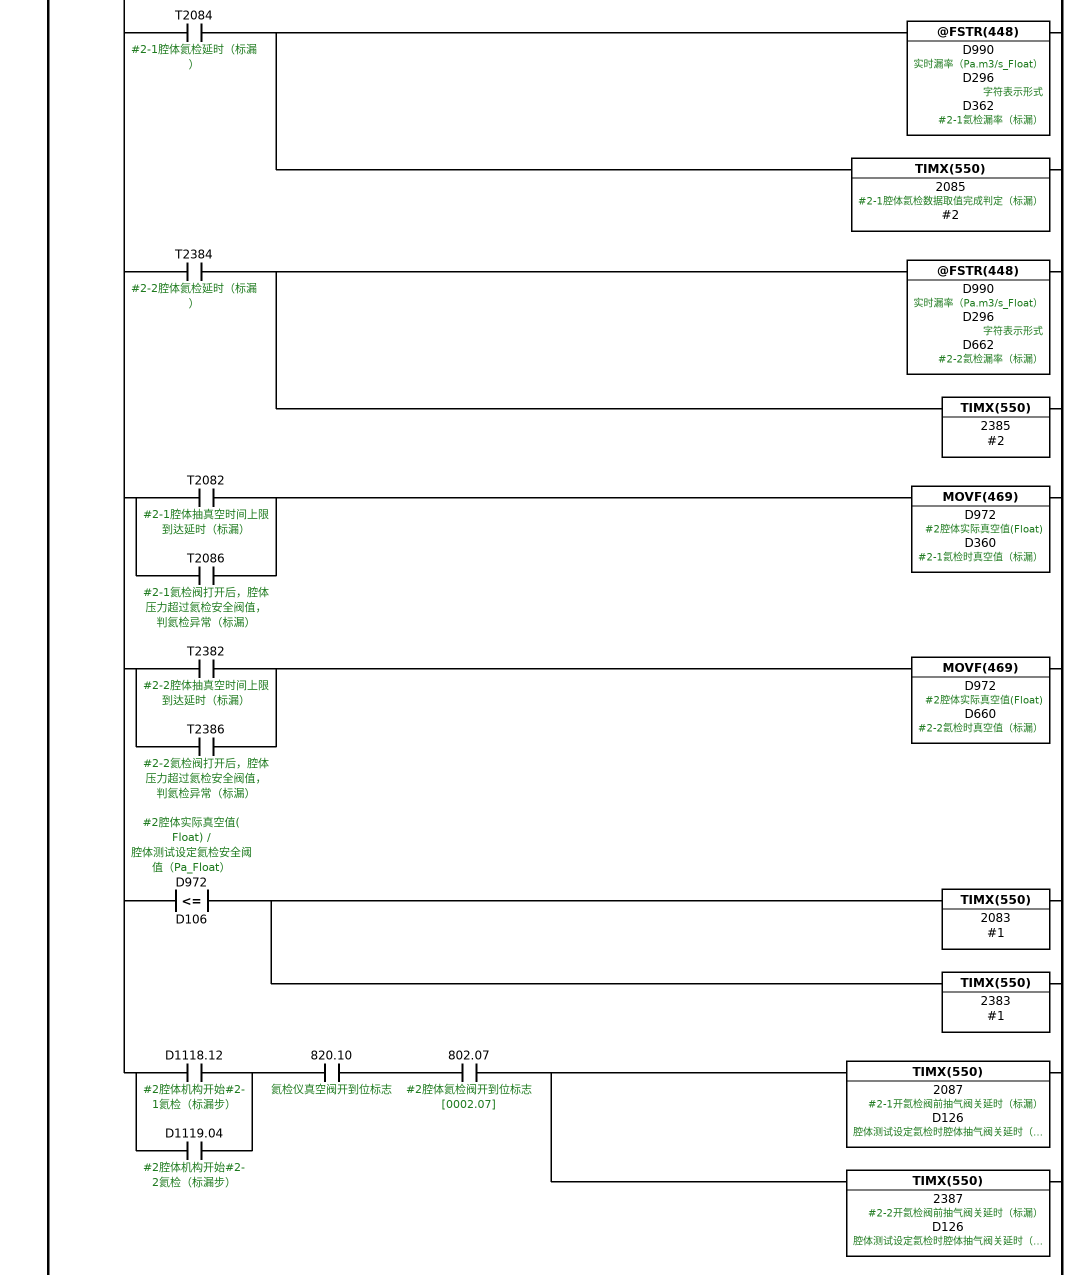
; rung 20: 标漏测试数据处理
LD P_On
OUT TR0
LD D1118.08  ; #2腔体机构开#2腔抽气阀（标漏步）
AND 821.10  ; #2-1腔体阀开到位标志
LD D1119.00  ; #2腔体机构开#2腔抽真空阀（标漏步）
AND 821.12  ; #2-2腔体阀开到位标志
ORLD
ANDLD
AND 821.08  ; #2腔体抽真空阀开到位标志
AND<=F(332) D972 D100  ; #2腔体实际真空值(Float), 腔体测试设定真空阈值（Pa_Float）
TIMX(550) 2081 #0  ; #2-1腔体抽真空阀值到达延时（标漏）
TIMX(550) 2381 #0  ; #2-2腔体抽真空阀值到达延时（标漏）
LD TR0
LD D1118.08  ; #2腔体机构开#2腔抽气阀（标漏步）
AND 821.10  ; #2-1腔体阀开到位标志
LD D1119.00  ; #2腔体机构开#2腔抽真空阀（标漏步）
AND 821.12  ; #2-2腔体阀开到位标志
ORLD
ANDLD
AND 821.08  ; #2腔体抽真空阀开到位标志
AND>F(333) D972 D100  ; #2腔体实际真空值(Float), 腔体测试设定真空阈值（Pa_Float）
TIMX(550) 2082 D102  ; 腔体测试设定抽真空时间上限（S_UInt）, #2-1腔体抽真空时间上限到达延时（标漏）
TIMX(550) 2382 D102  ; 腔体测试设定抽真空时间上限（S_UInt）, #2-2腔体抽真空时间上限到达延时（标漏）
LD TR0
AND D1118.12  ; #2腔体机构开始#2-1氦检（标漏步）
AND 821.10  ; #2-1腔体阀开到位标志
AND 820.10  ; 氦检仪真空阀开到位标志
AND 802.07  ; #2腔体氦检阀开到位标志[0002.07]
TIMX(550) 2084 D110  ; 腔体测试设定氦检时间（S_UInt）, #2-1腔体氦检延时（标漏）
@MOVF(469) D972 D360  ; #2腔体实际真空值(Float), #2-1氦检时真空值（标漏）
AND>F(333) D972 D106  ; #2腔体实际真空值(Float), 腔体测试设定氦检安全阈值（Pa_Float）
TIMX(550) 2086 #0  ; #2-1氦检阀打开后，腔体压力超过氦检安全阀值，判氦检异常（标漏）
LD TR0
AND D1119.04  ; #2腔体机构开始#2-2氦检（标漏步）
AND 821.12  ; #2-2腔体阀开到位标志
AND 820.10  ; 氦检仪真空阀开到位标志
AND 802.07  ; #2腔体氦检阀开到位标志[0002.07]
TIMX(550) 2384 D110  ; 腔体测试设定氦检时间（S_UInt）, #2-2腔体氦检延时（标漏）
@MOVF(469) D972 D660  ; #2腔体实际真空值(Float), #2-2氦检时真空值（标漏）
AND>F(333) D972 D106  ; #2腔体实际真空值(Float), 腔体测试设定氦检安全阈值（Pa_Float）
TIMX(550) 2386 #0  ; #2-2氦检阀打开后，腔体压力超过氦检安全阀值，判氦检异常（标漏）
LD TR0
AND T2084  ; #2-1腔体氦检延时（标漏）
@FSTR(448) D990 D296 D362  ; 实时漏率（Pa.m3/s_Float）, 字符表示形式, #2-1氦检漏率（标漏）
TIMX(550) 2085 #2  ; #2-1腔体氦检数据取值完成判定（标漏）
LD TR0
AND T2384  ; #2-2腔体氦检延时（标漏）
@FSTR(448) D990 D296 D662  ; 实时漏率（Pa.m3/s_Float）, 字符表示形式, #2-2氦检漏率（标漏）
TIMX(550) 2385 #2
LD TR0
LD T2082  ; #2-1腔体抽真空时间上限到达延时（标漏）
OR T2086  ; #2-1氦检阀打开后，腔体压力超过氦检安全阀值，判氦检异常（标漏）
ANDLD
MOVF(469) D972 D360  ; #2腔体实际真空值(Float), #2-1氦检时真空值（标漏）
LD TR0
LD T2382  ; #2-2腔体抽真空时间上限到达延时（标漏）
OR T2386  ; #2-2氦检阀打开后，腔体压力超过氦检安全阀值，判氦检异常（标漏）
ANDLD
MOVF(469) D972 D660  ; #2腔体实际真空值(Float), #2-2氦检时真空值（标漏）
LD TR0
AND<=F(332) D972 D106  ; #2腔体实际真空值(Float), 腔体测试设定氦检安全阈值（Pa_Float）
TIMX(550) 2083 #1
TIMX(550) 2383 #1
LD TR0
LD D1118.12  ; #2腔体机构开始#2-1氦检（标漏步）
OR D1119.04  ; #2腔体机构开始#2-2氦检（标漏步）
ANDLD
AND 820.10  ; 氦检仪真空阀开到位标志
AND 802.07  ; #2腔体氦检阀开到位标志[0002.07]
TIMX(550) 2087 D126  ; 腔体测试设定氦检时腔体抽气阀关延时（S_UInt）, #2-1开氦检阀前抽气阀关延时（标漏）
TIMX(550) 2387 D126  ; 腔体测试设定氦检时腔体抽气阀关延时（S_UInt）, #2-2开氦检阀前抽气阀关延时（标漏）
; rung 21: ********************** / #3腔体标漏流程 / **********************

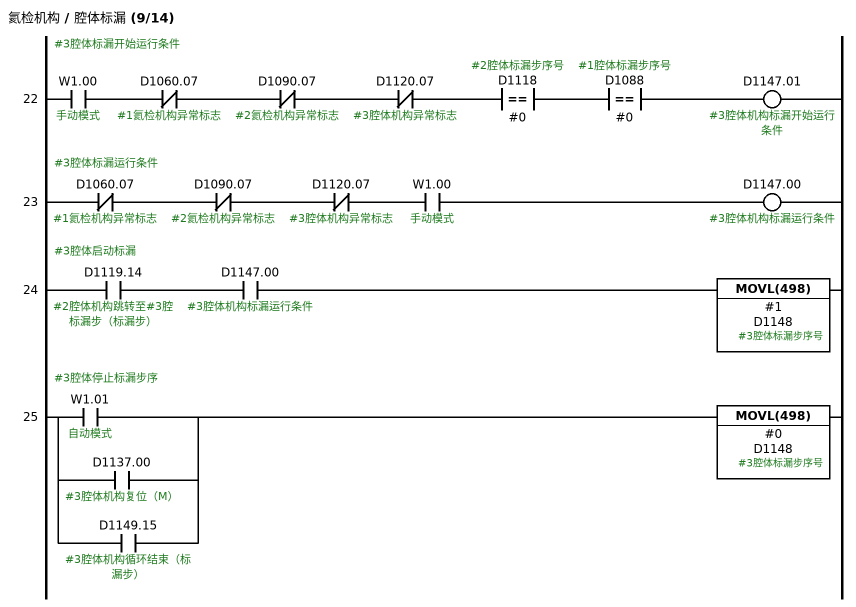
; rung 22: #3腔体标漏开始运行条件
LD W1.00  ; 手动模式
ANDNOT D1060.07  ; #1氦检机构异常标志
ANDNOT D1090.07  ; #2氦检机构异常标志
ANDNOT D1120.07  ; #3腔体机构异常标志
AND=L(301) D1118 #0  ; #2腔体标漏步序号
AND=L(301) D1088 #0  ; #1腔体标漏步序号
OUT D1147.01  ; #3腔体机构标漏开始运行条件
; rung 23: #3腔体标漏运行条件
LDNOT D1060.07  ; #1氦检机构异常标志
ANDNOT D1090.07  ; #2氦检机构异常标志
ANDNOT D1120.07  ; #3腔体机构异常标志
AND W1.00  ; 手动模式
OUT D1147.00  ; #3腔体机构标漏运行条件
; rung 24: #3腔体启动标漏
LD D1119.14  ; #2腔体机构跳转至#3腔标漏步（标漏步）
AND D1147.00  ; #3腔体机构标漏运行条件
MOVL(498) #1 D1148  ; #3腔体标漏步序号
; rung 25: #3腔体停止标漏步序
LD W1.01  ; 自动模式
OR D1137.00  ; #3腔体机构复位（M）
OR D1149.15  ; #3腔体机构循环结束（标漏步）
MOVL(498) #0 D1148  ; #3腔体标漏步序号

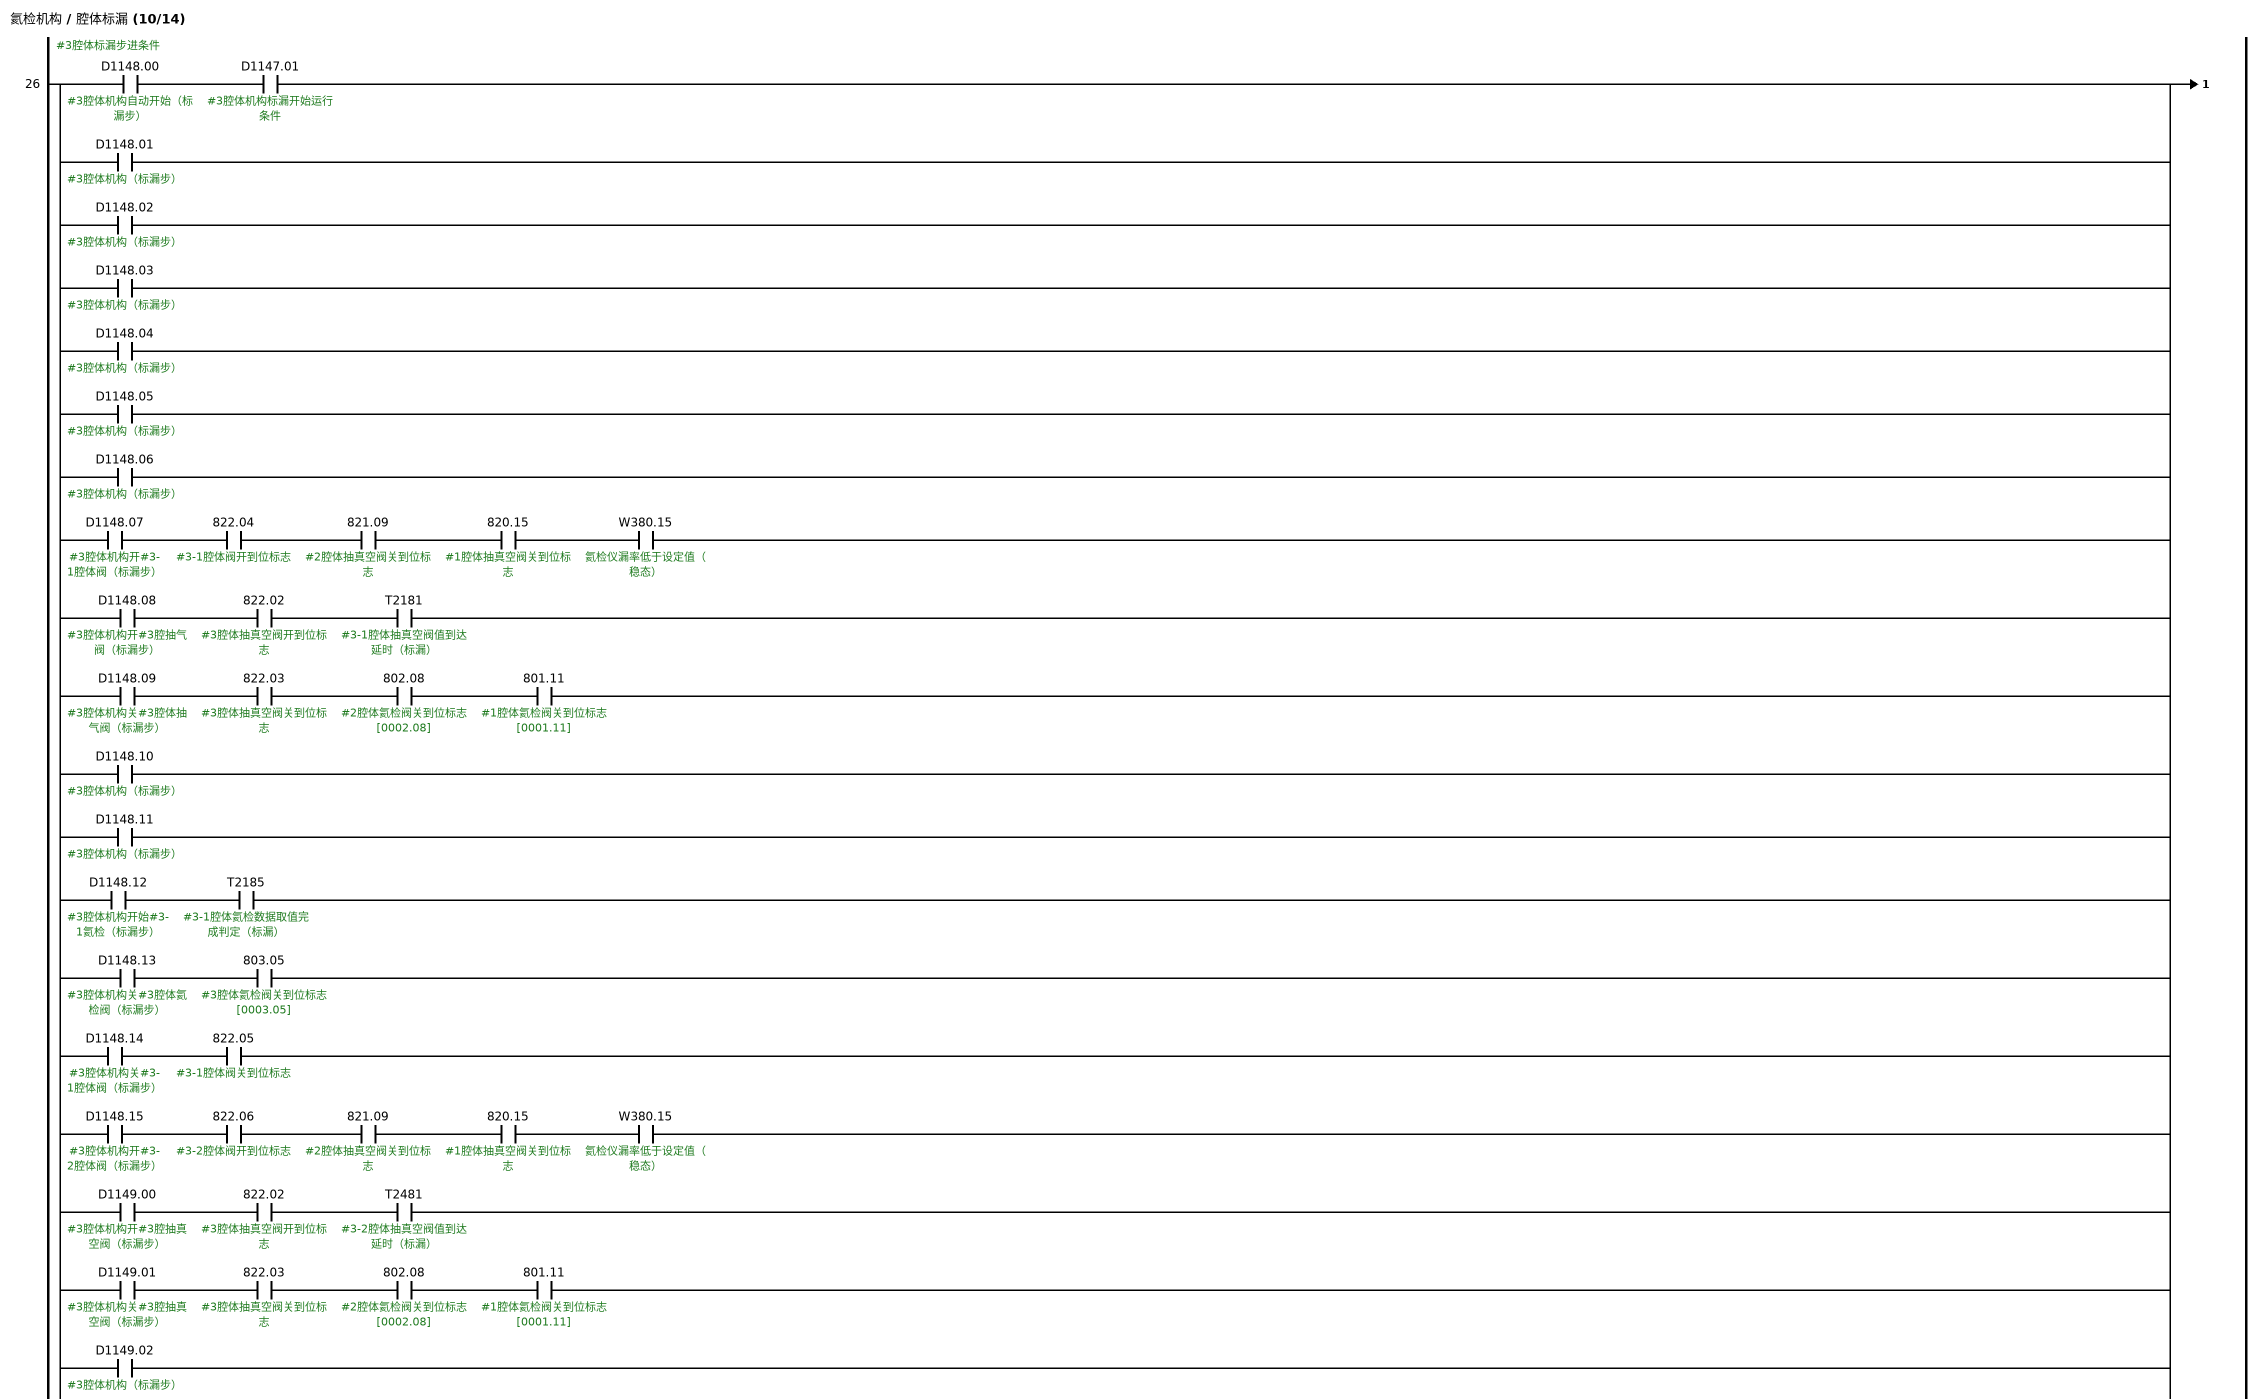

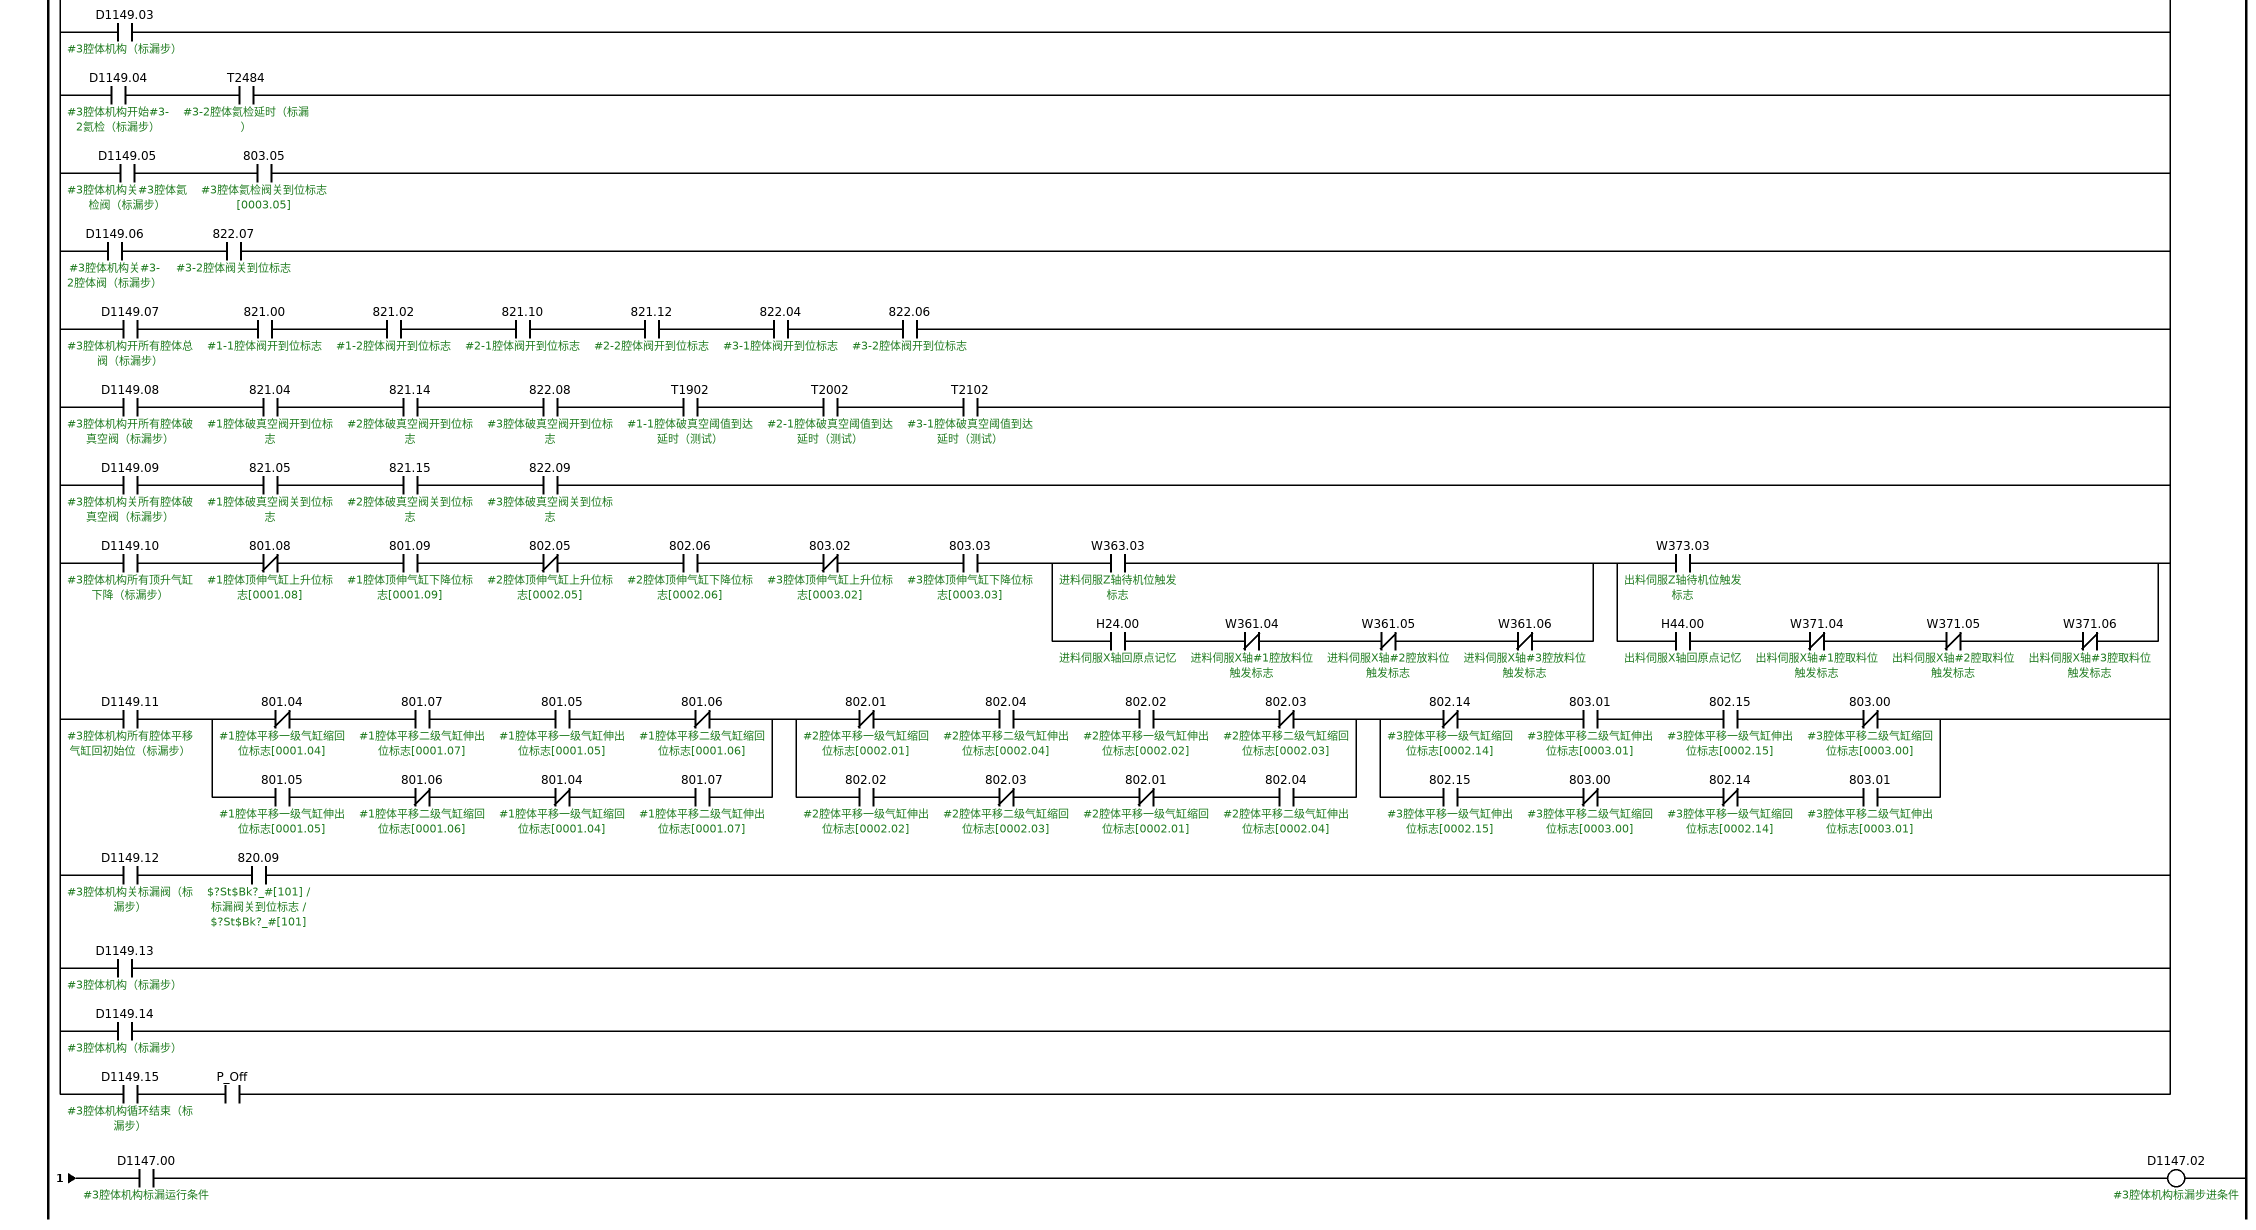
; rung 26: #3腔体标漏步进条件
LD D1148.00  ; #3腔体机构自动开始（标漏步）
AND D1147.01  ; #3腔体机构标漏开始运行条件
OR D1148.01  ; #3腔体机构（标漏步）
OR D1148.02  ; #3腔体机构（标漏步）
OR D1148.03  ; #3腔体机构（标漏步）
OR D1148.04  ; #3腔体机构（标漏步）
OR D1148.05  ; #3腔体机构（标漏步）
OR D1148.06  ; #3腔体机构（标漏步）
LD D1148.07  ; #3腔体机构开#3-1腔体阀（标漏步）
AND 822.04  ; #3-1腔体阀开到位标志
AND 821.09  ; #2腔体抽真空阀关到位标志
AND 820.15  ; #1腔体抽真空阀关到位标志
AND W380.15  ; 氦检仪漏率低于设定值（稳态）
ORLD
LD D1148.08  ; #3腔体机构开#3腔抽气阀（标漏步）
AND 822.02  ; #3腔体抽真空阀开到位标志
AND T2181  ; #3-1腔体抽真空阀值到达延时（标漏）
ORLD
LD D1148.09  ; #3腔体机构关#3腔体抽气阀（标漏步）
AND 822.03  ; #3腔体抽真空阀关到位标志
AND 802.08  ; #2腔体氦检阀关到位标志[0002.08]
AND 801.11  ; #1腔体氦检阀关到位标志[0001.11]
ORLD
OR D1148.10  ; #3腔体机构（标漏步）
OR D1148.11  ; #3腔体机构（标漏步）
LD D1148.12  ; #3腔体机构开始#3-1氦检（标漏步）
AND T2185  ; #3-1腔体氦检数据取值完成判定（标漏）
ORLD
LD D1148.13  ; #3腔体机构关#3腔体氦检阀（标漏步）
AND 803.05  ; #3腔体氦检阀关到位标志[0003.05]
ORLD
LD D1148.14  ; #3腔体机构关#3-1腔体阀（标漏步）
AND 822.05  ; #3-1腔体阀关到位标志
ORLD
LD D1148.15  ; #3腔体机构开#3-2腔体阀（标漏步）
AND 822.06  ; #3-2腔体阀开到位标志
AND 821.09  ; #2腔体抽真空阀关到位标志
AND 820.15  ; #1腔体抽真空阀关到位标志
AND W380.15  ; 氦检仪漏率低于设定值（稳态）
ORLD
LD D1149.00  ; #3腔体机构开#3腔抽真空阀（标漏步）
AND 822.02  ; #3腔体抽真空阀开到位标志
AND T2481  ; #3-2腔体抽真空阀值到达延时（标漏）
ORLD
LD D1149.01  ; #3腔体机构关#3腔抽真空阀（标漏步）
AND 822.03  ; #3腔体抽真空阀关到位标志
AND 802.08  ; #2腔体氦检阀关到位标志[0002.08]
AND 801.11  ; #1腔体氦检阀关到位标志[0001.11]
ORLD
OR D1149.02  ; #3腔体机构（标漏步）
OR D1149.03  ; #3腔体机构（标漏步）
LD D1149.04  ; #3腔体机构开始#3-2氦检（标漏步）
AND T2484  ; #3-2腔体氦检延时（标漏）
ORLD
LD D1149.05  ; #3腔体机构关#3腔体氦检阀（标漏步）
AND 803.05  ; #3腔体氦检阀关到位标志[0003.05]
ORLD
LD D1149.06  ; #3腔体机构关#3-2腔体阀（标漏步）
AND 822.07  ; #3-2腔体阀关到位标志
ORLD
LD D1149.07  ; #3腔体机构开所有腔体总阀（标漏步）
AND 821.00  ; #1-1腔体阀开到位标志
AND 821.02  ; #1-2腔体阀开到位标志
AND 821.10  ; #2-1腔体阀开到位标志
AND 821.12  ; #2-2腔体阀开到位标志
AND 822.04  ; #3-1腔体阀开到位标志
AND 822.06  ; #3-2腔体阀开到位标志
ORLD
LD D1149.08  ; #3腔体机构开所有腔体破真空阀（标漏步）
AND 821.04  ; #1腔体破真空阀开到位标志
AND 821.14  ; #2腔体破真空阀开到位标志
AND 822.08  ; #3腔体破真空阀开到位标志
AND T1902  ; #1-1腔体破真空阈值到达延时（测试）
AND T2002  ; #2-1腔体破真空阈值到达延时（测试）
AND T2102  ; #3-1腔体破真空阈值到达延时（测试）
ORLD
LD D1149.09  ; #3腔体机构关所有腔体破真空阀（标漏步）
AND 821.05  ; #1腔体破真空阀关到位标志
AND 821.15  ; #2腔体破真空阀关到位标志
AND 822.09  ; #3腔体破真空阀关到位标志
ORLD
LD D1149.10  ; #3腔体机构所有顶升气缸下降（标漏步）
ANDNOT 801.08  ; #1腔体顶伸气缸上升位标志[0001.08]
AND 801.09  ; #1腔体顶伸气缸下降位标志[0001.09]
ANDNOT 802.05  ; #2腔体顶伸气缸上升位标志[0002.05]
AND 802.06  ; #2腔体顶伸气缸下降位标志[0002.06]
ANDNOT 803.02  ; #3腔体顶伸气缸上升位标志[0003.02]
AND 803.03  ; #3腔体顶伸气缸下降位标志[0003.03]
LD W363.03  ; 进料伺服Z轴待机位触发标志
LD H24.00  ; 进料伺服X轴回原点记忆
ANDNOT W361.04  ; 进料伺服X轴#1腔放料位触发标志
ANDNOT W361.05  ; 进料伺服X轴#2腔放料位触发标志
ANDNOT W361.06  ; 进料伺服X轴#3腔放料位触发标志
ORLD
ANDLD
LD W373.03  ; 出料伺服Z轴待机位触发标志
LD H44.00  ; 出料伺服X轴回原点记忆
ANDNOT W371.04  ; 出料伺服X轴#1腔取料位触发标志
ANDNOT W371.05  ; 出料伺服X轴#2腔取料位触发标志
ANDNOT W371.06  ; 出料伺服X轴#3腔取料位触发标志
ORLD
ANDLD
ORLD
LD D1149.11  ; #3腔体机构所有腔体平移气缸回初始位（标漏步）
LDNOT 801.04  ; #1腔体平移一级气缸缩回位标志[0001.04]
AND 801.07  ; #1腔体平移二级气缸伸出位标志[0001.07]
AND 801.05  ; #1腔体平移一级气缸伸出位标志[0001.05]
ANDNOT 801.06  ; #1腔体平移二级气缸缩回位标志[0001.06]
LD 801.05  ; #1腔体平移一级气缸伸出位标志[0001.05]
ANDNOT 801.06  ; #1腔体平移二级气缸缩回位标志[0001.06]
ANDNOT 801.04  ; #1腔体平移一级气缸缩回位标志[0001.04]
AND 801.07  ; #1腔体平移二级气缸伸出位标志[0001.07]
ORLD
ANDLD
LDNOT 802.01  ; #2腔体平移一级气缸缩回位标志[0002.01]
AND 802.04  ; #2腔体平移二级气缸伸出位标志[0002.04]
AND 802.02  ; #2腔体平移一级气缸伸出位标志[0002.02]
ANDNOT 802.03  ; #2腔体平移二级气缸缩回位标志[0002.03]
LD 802.02  ; #2腔体平移一级气缸伸出位标志[0002.02]
ANDNOT 802.03  ; #2腔体平移二级气缸缩回位标志[0002.03]
ANDNOT 802.01  ; #2腔体平移一级气缸缩回位标志[0002.01]
AND 802.04  ; #2腔体平移二级气缸伸出位标志[0002.04]
ORLD
ANDLD
LDNOT 802.14  ; #3腔体平移一级气缸缩回位标志[0002.14]
AND 803.01  ; #3腔体平移二级气缸伸出位标志[0003.01]
AND 802.15  ; #3腔体平移一级气缸伸出位标志[0002.15]
ANDNOT 803.00  ; #3腔体平移二级气缸缩回位标志[0003.00]
LD 802.15  ; #3腔体平移一级气缸伸出位标志[0002.15]
ANDNOT 803.00  ; #3腔体平移二级气缸缩回位标志[0003.00]
ANDNOT 802.14  ; #3腔体平移一级气缸缩回位标志[0002.14]
AND 803.01  ; #3腔体平移二级气缸伸出位标志[0003.01]
ORLD
ANDLD
ORLD
LD D1149.12  ; #3腔体机构关标漏阀（标漏步）
AND 820.09  ; $?St$Bk?_#[101] / 标漏阀关到位标志 / $?St$Bk?_#[101]
ORLD
OR D1149.13  ; #3腔体机构（标漏步）
OR D1149.14  ; #3腔体机构（标漏步）
LD D1149.15  ; #3腔体机构循环结束（标漏步）
AND P_Off
ORLD
AND D1147.00  ; #3腔体机构标漏运行条件
OUT D1147.02  ; #3腔体机构标漏步进条件

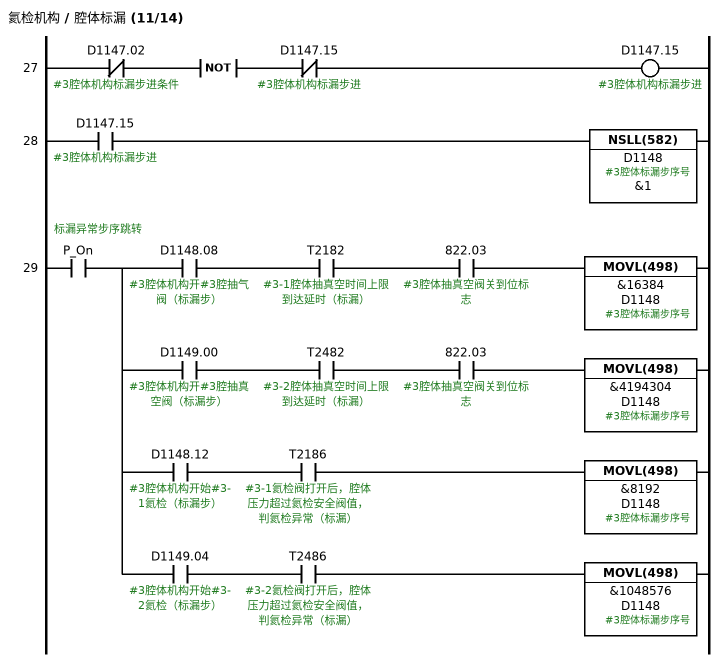
; rung 27
LDNOT D1147.02  ; #3腔体机构标漏步进条件
NOT(520)
ANDNOT D1147.15  ; #3腔体机构标漏步进
OUT D1147.15  ; #3腔体机构标漏步进
; rung 28
LD D1147.15  ; #3腔体机构标漏步进
NSLL(582) D1148 &1  ; #3腔体标漏步序号
; rung 29: 标漏异常步序跳转
LD P_On
OUT TR0
AND D1148.08  ; #3腔体机构开#3腔抽气阀（标漏步）
AND T2182  ; #3-1腔体抽真空时间上限到达延时（标漏）
AND 822.03  ; #3腔体抽真空阀关到位标志
MOVL(498) &16384 D1148  ; #3腔体标漏步序号
LD TR0
AND D1149.00  ; #3腔体机构开#3腔抽真空阀（标漏步）
AND T2482  ; #3-2腔体抽真空时间上限到达延时（标漏）
AND 822.03  ; #3腔体抽真空阀关到位标志
MOVL(498) &4194304 D1148  ; #3腔体标漏步序号
LD TR0
AND D1148.12  ; #3腔体机构开始#3-1氦检（标漏步）
AND T2186  ; #3-1氦检阀打开后，腔体压力超过氦检安全阀值，判氦检异常（标漏）
MOVL(498) &8192 D1148  ; #3腔体标漏步序号
LD TR0
AND D1149.04  ; #3腔体机构开始#3-2氦检（标漏步）
AND T2486  ; #3-2氦检阀打开后，腔体压力超过氦检安全阀值，判氦检异常（标漏）
MOVL(498) &1048576 D1148  ; #3腔体标漏步序号

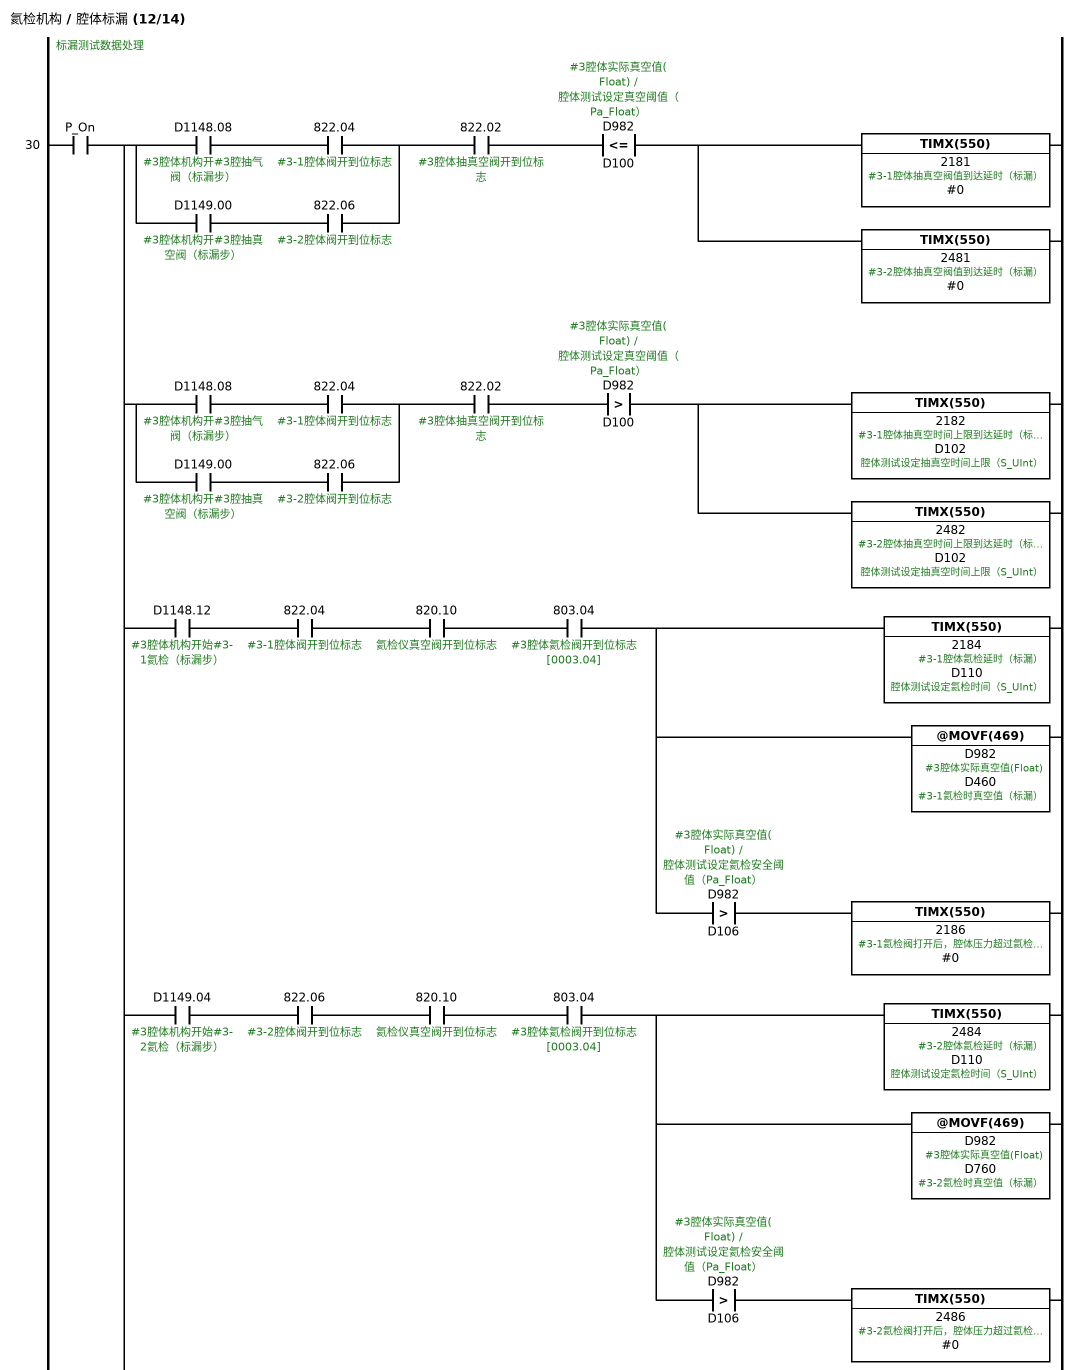

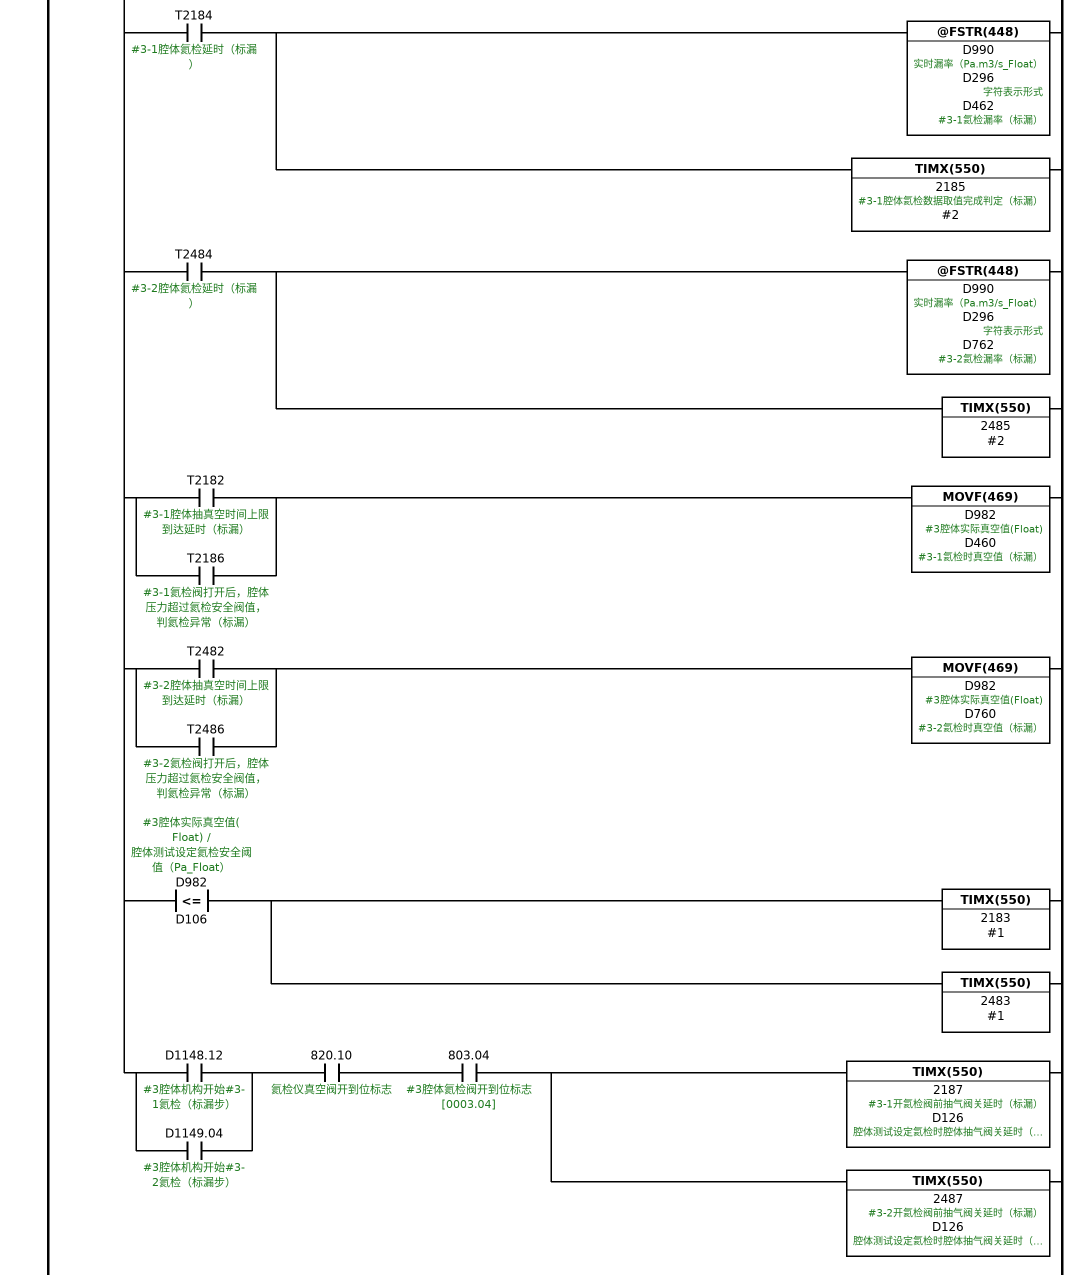
; rung 30: 标漏测试数据处理
LD P_On
OUT TR0
LD D1148.08  ; #3腔体机构开#3腔抽气阀（标漏步）
AND 822.04  ; #3-1腔体阀开到位标志
LD D1149.00  ; #3腔体机构开#3腔抽真空阀（标漏步）
AND 822.06  ; #3-2腔体阀开到位标志
ORLD
ANDLD
AND 822.02  ; #3腔体抽真空阀开到位标志
AND<=F(332) D982 D100  ; #3腔体实际真空值(Float), 腔体测试设定真空阈值（Pa_Float）
TIMX(550) 2181 #0  ; #3-1腔体抽真空阀值到达延时（标漏）
TIMX(550) 2481 #0  ; #3-2腔体抽真空阀值到达延时（标漏）
LD TR0
LD D1148.08  ; #3腔体机构开#3腔抽气阀（标漏步）
AND 822.04  ; #3-1腔体阀开到位标志
LD D1149.00  ; #3腔体机构开#3腔抽真空阀（标漏步）
AND 822.06  ; #3-2腔体阀开到位标志
ORLD
ANDLD
AND 822.02  ; #3腔体抽真空阀开到位标志
AND>F(333) D982 D100  ; #3腔体实际真空值(Float), 腔体测试设定真空阈值（Pa_Float）
TIMX(550) 2182 D102  ; 腔体测试设定抽真空时间上限（S_UInt）, #3-1腔体抽真空时间上限到达延时（标漏）
TIMX(550) 2482 D102  ; 腔体测试设定抽真空时间上限（S_UInt）, #3-2腔体抽真空时间上限到达延时（标漏）
LD TR0
AND D1148.12  ; #3腔体机构开始#3-1氦检（标漏步）
AND 822.04  ; #3-1腔体阀开到位标志
AND 820.10  ; 氦检仪真空阀开到位标志
AND 803.04  ; #3腔体氦检阀开到位标志[0003.04]
TIMX(550) 2184 D110  ; 腔体测试设定氦检时间（S_UInt）, #3-1腔体氦检延时（标漏）
@MOVF(469) D982 D460  ; #3腔体实际真空值(Float), #3-1氦检时真空值（标漏）
AND>F(333) D982 D106  ; #3腔体实际真空值(Float), 腔体测试设定氦检安全阈值（Pa_Float）
TIMX(550) 2186 #0  ; #3-1氦检阀打开后，腔体压力超过氦检安全阀值，判氦检异常（标漏）
LD TR0
AND D1149.04  ; #3腔体机构开始#3-2氦检（标漏步）
AND 822.06  ; #3-2腔体阀开到位标志
AND 820.10  ; 氦检仪真空阀开到位标志
AND 803.04  ; #3腔体氦检阀开到位标志[0003.04]
TIMX(550) 2484 D110  ; 腔体测试设定氦检时间（S_UInt）, #3-2腔体氦检延时（标漏）
@MOVF(469) D982 D760  ; #3腔体实际真空值(Float), #3-2氦检时真空值（标漏）
AND>F(333) D982 D106  ; #3腔体实际真空值(Float), 腔体测试设定氦检安全阈值（Pa_Float）
TIMX(550) 2486 #0  ; #3-2氦检阀打开后，腔体压力超过氦检安全阀值，判氦检异常（标漏）
LD TR0
AND T2184  ; #3-1腔体氦检延时（标漏）
@FSTR(448) D990 D296 D462  ; 实时漏率（Pa.m3/s_Float）, 字符表示形式, #3-1氦检漏率（标漏）
TIMX(550) 2185 #2  ; #3-1腔体氦检数据取值完成判定（标漏）
LD TR0
AND T2484  ; #3-2腔体氦检延时（标漏）
@FSTR(448) D990 D296 D762  ; 实时漏率（Pa.m3/s_Float）, 字符表示形式, #3-2氦检漏率（标漏）
TIMX(550) 2485 #2
LD TR0
LD T2182  ; #3-1腔体抽真空时间上限到达延时（标漏）
OR T2186  ; #3-1氦检阀打开后，腔体压力超过氦检安全阀值，判氦检异常（标漏）
ANDLD
MOVF(469) D982 D460  ; #3腔体实际真空值(Float), #3-1氦检时真空值（标漏）
LD TR0
LD T2482  ; #3-2腔体抽真空时间上限到达延时（标漏）
OR T2486  ; #3-2氦检阀打开后，腔体压力超过氦检安全阀值，判氦检异常（标漏）
ANDLD
MOVF(469) D982 D760  ; #3腔体实际真空值(Float), #3-2氦检时真空值（标漏）
LD TR0
AND<=F(332) D982 D106  ; #3腔体实际真空值(Float), 腔体测试设定氦检安全阈值（Pa_Float）
TIMX(550) 2183 #1
TIMX(550) 2483 #1
LD TR0
LD D1148.12  ; #3腔体机构开始#3-1氦检（标漏步）
OR D1149.04  ; #3腔体机构开始#3-2氦检（标漏步）
ANDLD
AND 820.10  ; 氦检仪真空阀开到位标志
AND 803.04  ; #3腔体氦检阀开到位标志[0003.04]
TIMX(550) 2187 D126  ; 腔体测试设定氦检时腔体抽气阀关延时（S_UInt）, #3-1开氦检阀前抽气阀关延时（标漏）
TIMX(550) 2487 D126  ; 腔体测试设定氦检时腔体抽气阀关延时（S_UInt）, #3-2开氦检阀前抽气阀关延时（标漏）

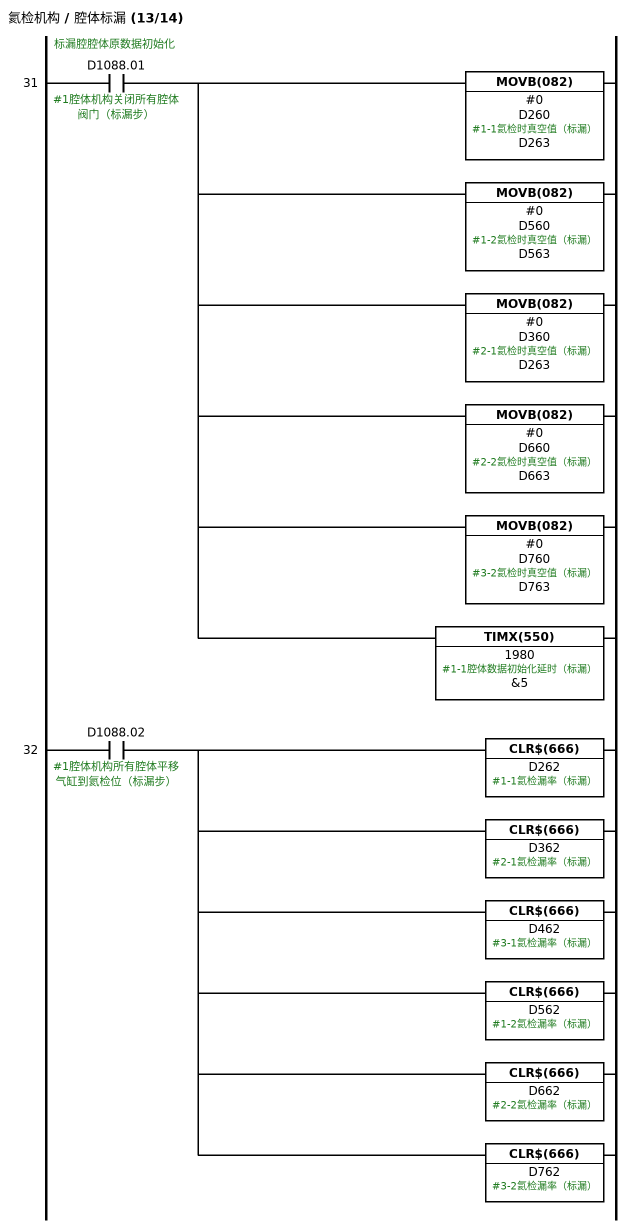
; rung 31: 标漏腔腔体原数据初始化
LD D1088.01  ; #1腔体机构关闭所有腔体阀门（标漏步）
MOVB(082) #0 D260 D263  ; #1-1氦检时真空值（标漏）
MOVB(082) #0 D560 D563  ; #1-2氦检时真空值（标漏）
MOVB(082) #0 D360 D263  ; #2-1氦检时真空值（标漏）
MOVB(082) #0 D660 D663  ; #2-2氦检时真空值（标漏）
MOVB(082) #0 D760 D763  ; #3-2氦检时真空值（标漏）
TIMX(550) 1980 &5  ; #1-1腔体数据初始化延时（标漏）
; rung 32
LD D1088.02  ; #1腔体机构所有腔体平移气缸到氦检位（标漏步）
CLR$(666) D262  ; #1-1氦检漏率（标漏）
CLR$(666) D362  ; #2-1氦检漏率（标漏）
CLR$(666) D462  ; #3-1氦检漏率（标漏）
CLR$(666) D562  ; #1-2氦检漏率（标漏）
CLR$(666) D662  ; #2-2氦检漏率（标漏）
CLR$(666) D762  ; #3-2氦检漏率（标漏）

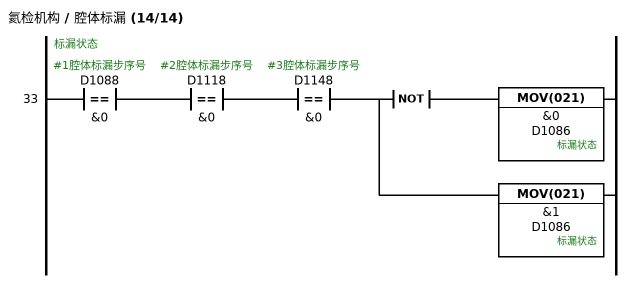
; rung 33: 标漏状态
LD=L(301) D1088 &0  ; #1腔体标漏步序号
AND=L(301) D1118 &0  ; #2腔体标漏步序号
AND=L(301) D1148 &0  ; #3腔体标漏步序号
OUT TR0
NOT(520)
MOV(021) &0 D1086  ; 标漏状态
LD TR0
MOV(021) &1 D1086  ; 标漏状态

### Section 腔体自检

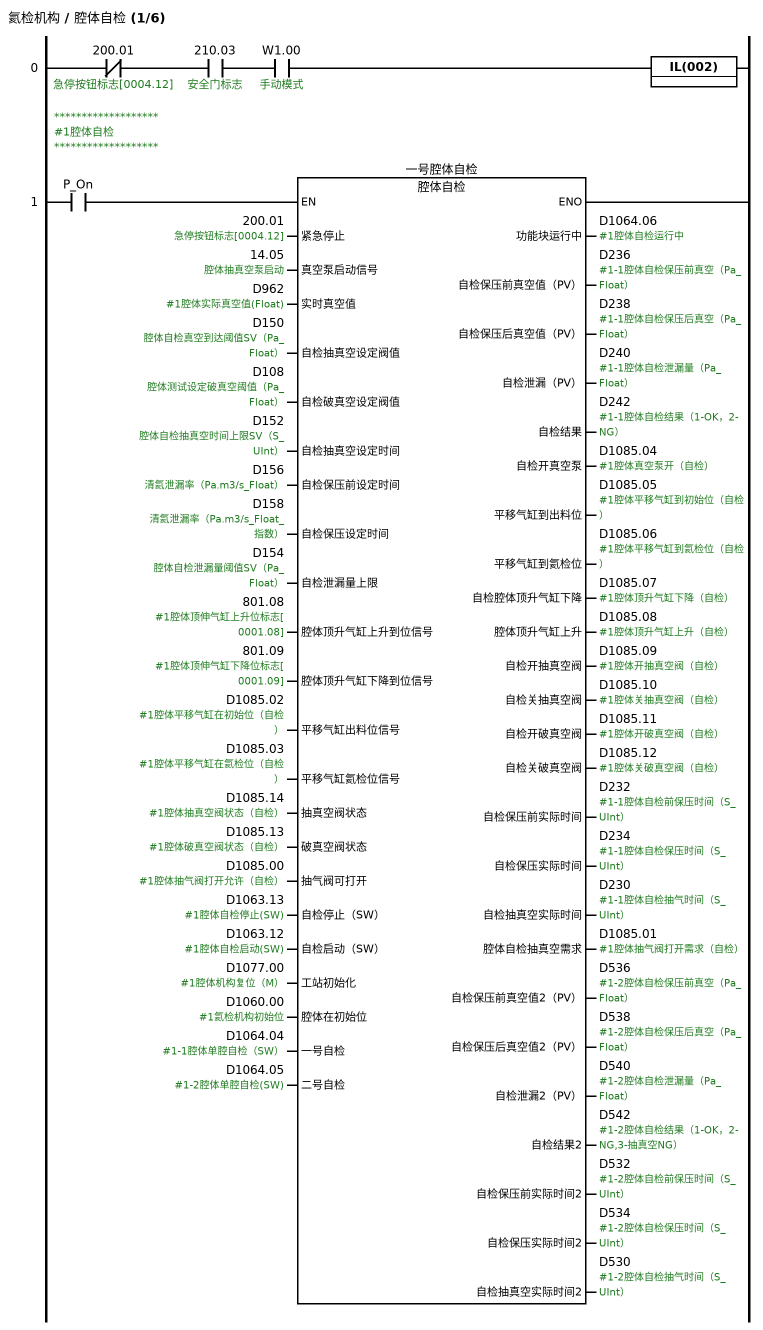
; rung 0
LDNOT 200.01  ; 急停按钮标志[0004.12]
AND 210.03  ; 安全门标志
AND W1.00  ; 手动模式
IL(002)
; rung 1: ******************* / #1腔体自检 / *******************
LD P_On
CALL 一号腔体自检 : 腔体自检 (紧急停止 := 200.01, 真空泵启动信号 := 14.05, 实时真空值 := D962, 自检抽真空设定阀值 := D150, 自检破真空设定阀值 := D108, 自检抽真空设定时间 := D152, 自检保压前设定时间 := D156, 自检保压设定时间 := D158, 自检泄漏量上限 := D154, 腔体顶升气缸上升到位信号 := 801.08, 腔体顶升气缸下降到位信号 := 801.09, 平移气缸出料位信号 := D1085.02, 平移气缸氦检位信号 := D1085.03, 抽真空阀状态 := D1085.14, 破真空阀状态 := D1085.13, 抽气阀可打开 := D1085.00, 自检停止（SW） := D1063.13, 自检启动（SW） := D1063.12, 工站初始化 := D1077.00, 腔体在初始位 := D1060.00, 一号自检 := D1064.04, 二号自检 := D1064.05, 功能块运行中 => D1064.06, 自检保压前真空值（PV） => D236, 自检保压后真空值（PV） => D238, 自检泄漏（PV） => D240, 自检结果 => D242, 自检开真空泵 => D1085.04, 平移气缸到出料位 => D1085.05, 平移气缸到氦检位 => D1085.06, 自检腔体顶升气缸下降 => D1085.07, 腔体顶升气缸上升 => D1085.08, 自检开抽真空阀 => D1085.09, 自检关抽真空阀 => D1085.10, 自检开破真空阀 => D1085.11, 自检关破真空阀 => D1085.12, 自检保压前实际时间 => D232, 自检保压实际时间 => D234, 自检抽真空实际时间 => D230, 腔体自检抽真空需求 => D1085.01, 自检保压前真空值2（PV） => D536, 自检保压后真空值2（PV） => D538, 自检泄漏2（PV） => D540, 自检结果2 => D542, 自检保压前实际时间2 => D532, 自检保压实际时间2 => D534, 自检抽真空实际时间2 => D530)  ; 急停按钮标志[0004.12], 腔体抽真空泵启动, #1腔体实际真空值(Float), 腔体自检真空到达阈值SV（Pa_Float）, 腔体测试设定破真空阈值（Pa_Float）, 腔体自检抽真空时间上限SV（S_UInt）, 清氦泄漏率（Pa.m3/s_Float）, 清氦泄漏率（Pa.m3/s_Float_指数）, 腔体自检泄漏量阈值SV（Pa_Float）, #1腔体顶伸气缸上升位标志[0001.08], #1腔体顶伸气缸下降位标志[0001.09], #1腔体平移气缸在初始位（自检）, #1腔体平移气缸在氦检位（自检）, #1腔体抽真空阀状态（自检）, #1腔体破真空阀状态（自检）, #1腔体抽气阀打开允许（自检）, #1腔体自检停止(SW), #1腔体自检启动(SW), #1腔体机构复位（M）, #1氦检机构初始位, #1-1腔体单腔自检（SW）, #1-2腔体单腔自检(SW), #1腔体自检运行中, #1-1腔体自检保压前真空（Pa_Float）, #1-1腔体自检保压后真空（Pa_Float）, #1-1腔体自检泄漏量（Pa_Float）, #1-1腔体自检结果（1-OK，2-NG）, #1腔体真空泵开（自检）, #1腔体平移气缸到初始位（自检）, #1腔体平移气缸到氦检位（自检）, #1腔体顶升气缸下降（自检）, #1腔体顶升气缸上升（自检）, #1腔体开抽真空阀（自检）, #1腔体关抽真空阀（自检）, #1腔体开破真空阀（自检）, #1腔体关破真空阀（自检）, #1-1腔体自检前保压时间（S_UInt）, #1-1腔体自检保压时间（S_UInt）, #1-1腔体自检抽气时间（S_UInt）, #1腔体抽气阀打开需求（自检）, #1-2腔体自检保压前真空（Pa_Float）, #1-2腔体自检保压后真空（Pa_Float）, #1-2腔体自检泄漏量（Pa_Float）, #1-2腔体自检结果（1-OK，2-NG,3-抽真空NG）, #1-2腔体自检前保压时间（S_UInt）, #1-2腔体自检保压时间（S_UInt）, #1-2腔体自检抽气时间（S_UInt）

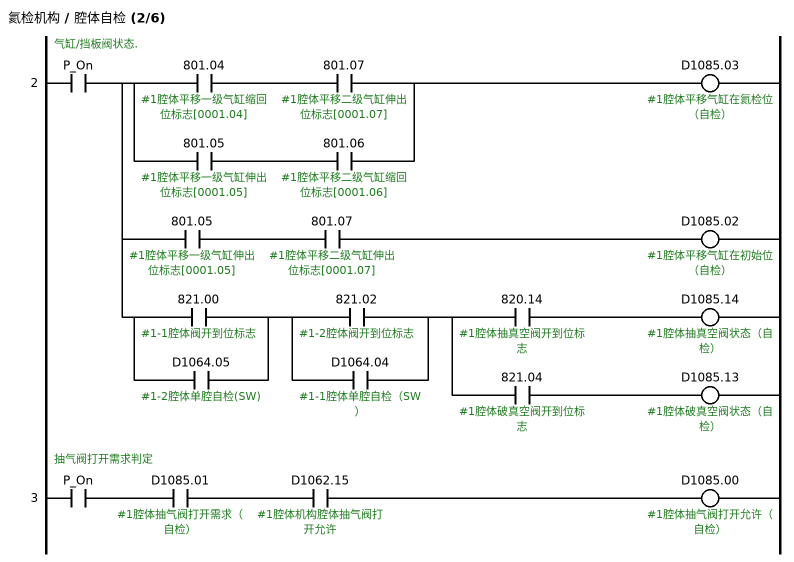
; rung 2: 气缸/挡板阀状态.
LD P_On
OUT TR0
LD 801.04  ; #1腔体平移一级气缸缩回位标志[0001.04]
AND 801.07  ; #1腔体平移二级气缸伸出位标志[0001.07]
LD 801.05  ; #1腔体平移一级气缸伸出位标志[0001.05]
AND 801.06  ; #1腔体平移二级气缸缩回位标志[0001.06]
ORLD
ANDLD
OUT D1085.03  ; #1腔体平移气缸在氦检位（自检）
LD TR0
AND 801.05  ; #1腔体平移一级气缸伸出位标志[0001.05]
AND 801.07  ; #1腔体平移二级气缸伸出位标志[0001.07]
OUT D1085.02  ; #1腔体平移气缸在初始位（自检）
LD TR0
LD 821.00  ; #1-1腔体阀开到位标志
OR D1064.05  ; #1-2腔体单腔自检(SW)
ANDLD
LD 821.02  ; #1-2腔体阀开到位标志
OR D1064.04  ; #1-1腔体单腔自检（SW）
ANDLD
OUT TR0
AND 820.14  ; #1腔体抽真空阀开到位标志
OUT D1085.14  ; #1腔体抽真空阀状态（自检）
LD TR0
AND 821.04  ; #1腔体破真空阀开到位标志
OUT D1085.13  ; #1腔体破真空阀状态（自检）
; rung 3: 抽气阀打开需求判定
LD P_On
AND D1085.01  ; #1腔体抽气阀打开需求（自检）
AND D1062.15  ; #1腔体机构腔体抽气阀打开允许
OUT D1085.00  ; #1腔体抽气阀打开允许（自检）

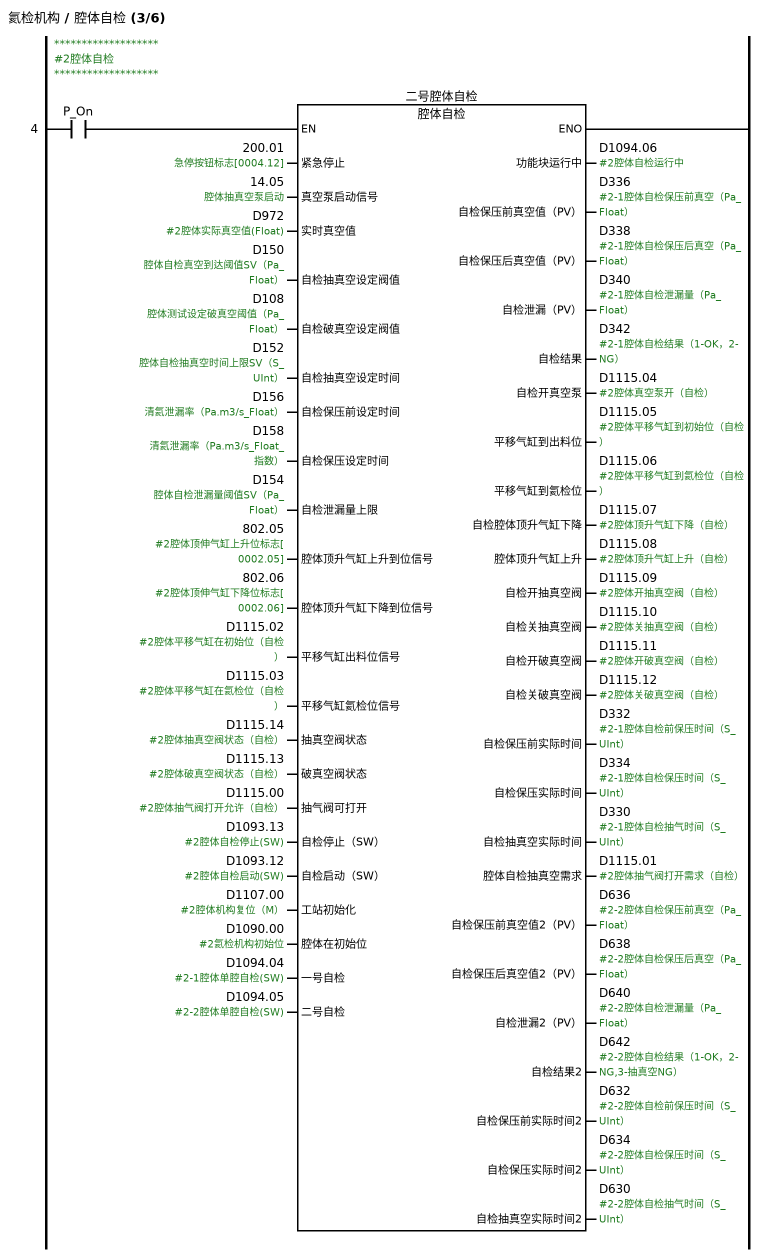
; rung 4: ******************* / #2腔体自检 / *******************
LD P_On
CALL 二号腔体自检 : 腔体自检 (紧急停止 := 200.01, 真空泵启动信号 := 14.05, 实时真空值 := D972, 自检抽真空设定阀值 := D150, 自检破真空设定阀值 := D108, 自检抽真空设定时间 := D152, 自检保压前设定时间 := D156, 自检保压设定时间 := D158, 自检泄漏量上限 := D154, 腔体顶升气缸上升到位信号 := 802.05, 腔体顶升气缸下降到位信号 := 802.06, 平移气缸出料位信号 := D1115.02, 平移气缸氦检位信号 := D1115.03, 抽真空阀状态 := D1115.14, 破真空阀状态 := D1115.13, 抽气阀可打开 := D1115.00, 自检停止（SW） := D1093.13, 自检启动（SW） := D1093.12, 工站初始化 := D1107.00, 腔体在初始位 := D1090.00, 一号自检 := D1094.04, 二号自检 := D1094.05, 功能块运行中 => D1094.06, 自检保压前真空值（PV） => D336, 自检保压后真空值（PV） => D338, 自检泄漏（PV） => D340, 自检结果 => D342, 自检开真空泵 => D1115.04, 平移气缸到出料位 => D1115.05, 平移气缸到氦检位 => D1115.06, 自检腔体顶升气缸下降 => D1115.07, 腔体顶升气缸上升 => D1115.08, 自检开抽真空阀 => D1115.09, 自检关抽真空阀 => D1115.10, 自检开破真空阀 => D1115.11, 自检关破真空阀 => D1115.12, 自检保压前实际时间 => D332, 自检保压实际时间 => D334, 自检抽真空实际时间 => D330, 腔体自检抽真空需求 => D1115.01, 自检保压前真空值2（PV） => D636, 自检保压后真空值2（PV） => D638, 自检泄漏2（PV） => D640, 自检结果2 => D642, 自检保压前实际时间2 => D632, 自检保压实际时间2 => D634, 自检抽真空实际时间2 => D630)  ; 急停按钮标志[0004.12], 腔体抽真空泵启动, #2腔体实际真空值(Float), 腔体自检真空到达阈值SV（Pa_Float）, 腔体测试设定破真空阈值（Pa_Float）, 腔体自检抽真空时间上限SV（S_UInt）, 清氦泄漏率（Pa.m3/s_Float）, 清氦泄漏率（Pa.m3/s_Float_指数）, 腔体自检泄漏量阈值SV（Pa_Float）, #2腔体顶伸气缸上升位标志[0002.05], #2腔体顶伸气缸下降位标志[0002.06], #2腔体平移气缸在初始位（自检）, #2腔体平移气缸在氦检位（自检）, #2腔体抽真空阀状态（自检）, #2腔体破真空阀状态（自检）, #2腔体抽气阀打开允许（自检）, #2腔体自检停止(SW), #2腔体自检启动(SW), #2腔体机构复位（M）, #2氦检机构初始位, #2-1腔体单腔自检(SW), #2-2腔体单腔自检(SW), #2腔体自检运行中, #2-1腔体自检保压前真空（Pa_Float）, #2-1腔体自检保压后真空（Pa_Float）, #2-1腔体自检泄漏量（Pa_Float）, #2-1腔体自检结果（1-OK，2-NG）, #2腔体真空泵开（自检）, #2腔体平移气缸到初始位（自检）, #2腔体平移气缸到氦检位（自检）, #2腔体顶升气缸下降（自检）, #2腔体顶升气缸上升（自检）, #2腔体开抽真空阀（自检）, #2腔体关抽真空阀（自检）, #2腔体开破真空阀（自检）, #2腔体关破真空阀（自检）, #2-1腔体自检前保压时间（S_UInt）, #2-1腔体自检保压时间（S_UInt）, #2-1腔体自检抽气时间（S_UInt）, #2腔体抽气阀打开需求（自检）, #2-2腔体自检保压前真空（Pa_Float）, #2-2腔体自检保压后真空（Pa_Float）, #2-2腔体自检泄漏量（Pa_Float）, #2-2腔体自检结果（1-OK，2-NG,3-抽真空NG）, #2-2腔体自检前保压时间（S_UInt）, #2-2腔体自检保压时间（S_UInt）, #2-2腔体自检抽气时间（S_UInt）

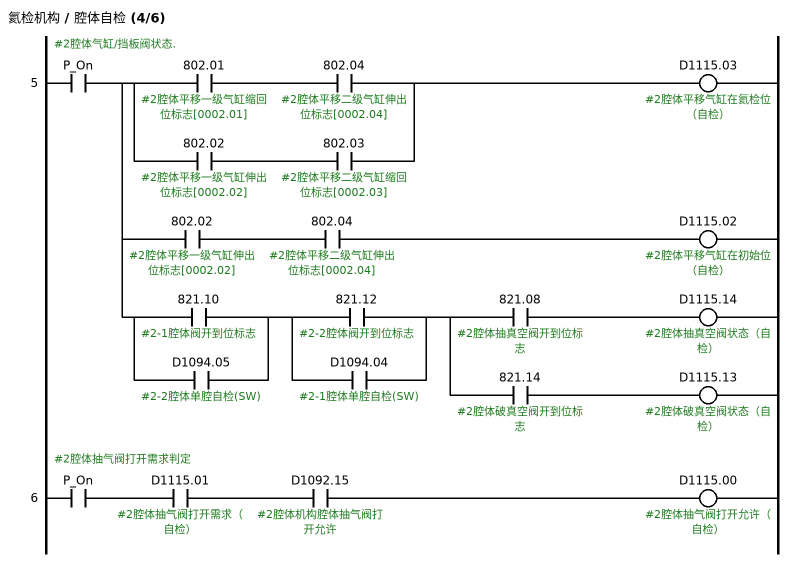
; rung 5: #2腔体气缸/挡板阀状态.
LD P_On
OUT TR0
LD 802.01  ; #2腔体平移一级气缸缩回位标志[0002.01]
AND 802.04  ; #2腔体平移二级气缸伸出位标志[0002.04]
LD 802.02  ; #2腔体平移一级气缸伸出位标志[0002.02]
AND 802.03  ; #2腔体平移二级气缸缩回位标志[0002.03]
ORLD
ANDLD
OUT D1115.03  ; #2腔体平移气缸在氦检位（自检）
LD TR0
AND 802.02  ; #2腔体平移一级气缸伸出位标志[0002.02]
AND 802.04  ; #2腔体平移二级气缸伸出位标志[0002.04]
OUT D1115.02  ; #2腔体平移气缸在初始位（自检）
LD TR0
LD 821.10  ; #2-1腔体阀开到位标志
OR D1094.05  ; #2-2腔体单腔自检(SW)
ANDLD
LD 821.12  ; #2-2腔体阀开到位标志
OR D1094.04  ; #2-1腔体单腔自检(SW)
ANDLD
OUT TR0
AND 821.08  ; #2腔体抽真空阀开到位标志
OUT D1115.14  ; #2腔体抽真空阀状态（自检）
LD TR0
AND 821.14  ; #2腔体破真空阀开到位标志
OUT D1115.13  ; #2腔体破真空阀状态（自检）
; rung 6: #2腔体抽气阀打开需求判定
LD P_On
AND D1115.01  ; #2腔体抽气阀打开需求（自检）
AND D1092.15  ; #2腔体机构腔体抽气阀打开允许
OUT D1115.00  ; #2腔体抽气阀打开允许（自检）

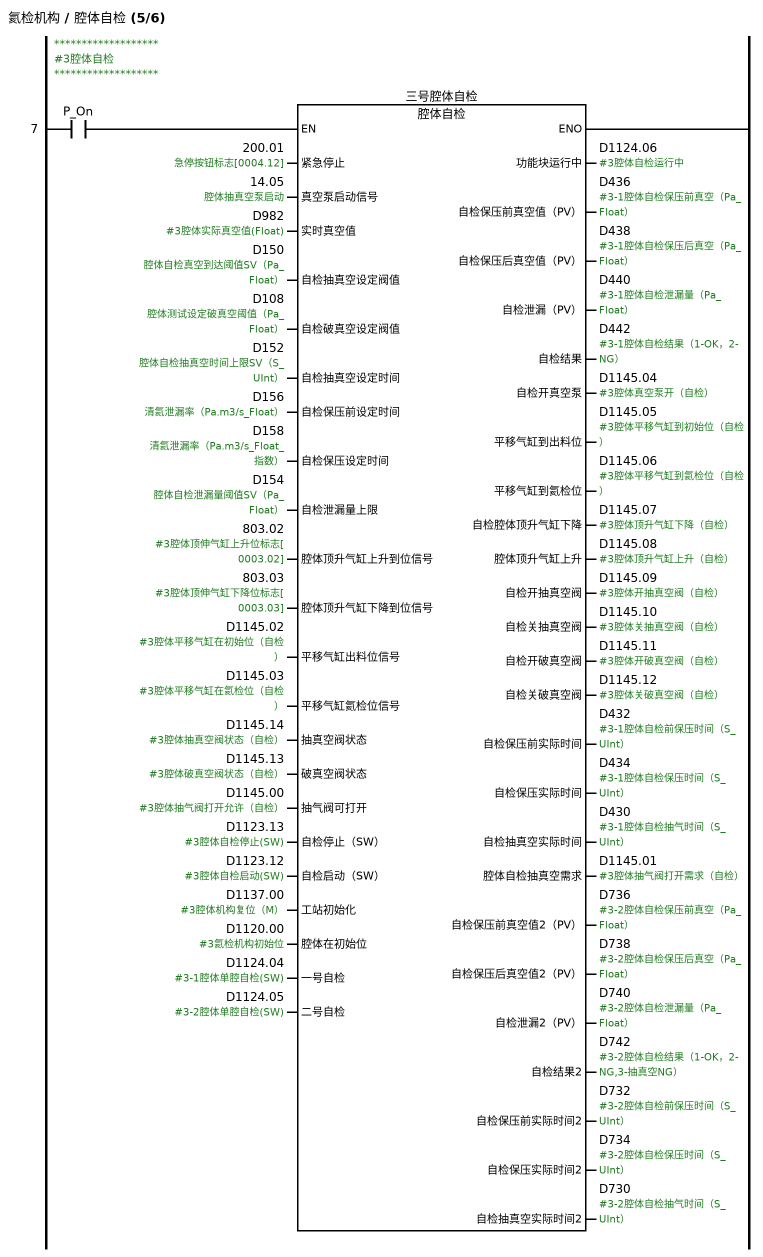
; rung 7: ******************* / #3腔体自检 / *******************
LD P_On
CALL 三号腔体自检 : 腔体自检 (紧急停止 := 200.01, 真空泵启动信号 := 14.05, 实时真空值 := D982, 自检抽真空设定阀值 := D150, 自检破真空设定阀值 := D108, 自检抽真空设定时间 := D152, 自检保压前设定时间 := D156, 自检保压设定时间 := D158, 自检泄漏量上限 := D154, 腔体顶升气缸上升到位信号 := 803.02, 腔体顶升气缸下降到位信号 := 803.03, 平移气缸出料位信号 := D1145.02, 平移气缸氦检位信号 := D1145.03, 抽真空阀状态 := D1145.14, 破真空阀状态 := D1145.13, 抽气阀可打开 := D1145.00, 自检停止（SW） := D1123.13, 自检启动（SW） := D1123.12, 工站初始化 := D1137.00, 腔体在初始位 := D1120.00, 一号自检 := D1124.04, 二号自检 := D1124.05, 功能块运行中 => D1124.06, 自检保压前真空值（PV） => D436, 自检保压后真空值（PV） => D438, 自检泄漏（PV） => D440, 自检结果 => D442, 自检开真空泵 => D1145.04, 平移气缸到出料位 => D1145.05, 平移气缸到氦检位 => D1145.06, 自检腔体顶升气缸下降 => D1145.07, 腔体顶升气缸上升 => D1145.08, 自检开抽真空阀 => D1145.09, 自检关抽真空阀 => D1145.10, 自检开破真空阀 => D1145.11, 自检关破真空阀 => D1145.12, 自检保压前实际时间 => D432, 自检保压实际时间 => D434, 自检抽真空实际时间 => D430, 腔体自检抽真空需求 => D1145.01, 自检保压前真空值2（PV） => D736, 自检保压后真空值2（PV） => D738, 自检泄漏2（PV） => D740, 自检结果2 => D742, 自检保压前实际时间2 => D732, 自检保压实际时间2 => D734, 自检抽真空实际时间2 => D730)  ; 急停按钮标志[0004.12], 腔体抽真空泵启动, #3腔体实际真空值(Float), 腔体自检真空到达阈值SV（Pa_Float）, 腔体测试设定破真空阈值（Pa_Float）, 腔体自检抽真空时间上限SV（S_UInt）, 清氦泄漏率（Pa.m3/s_Float）, 清氦泄漏率（Pa.m3/s_Float_指数）, 腔体自检泄漏量阈值SV（Pa_Float）, #3腔体顶伸气缸上升位标志[0003.02], #3腔体顶伸气缸下降位标志[0003.03], #3腔体平移气缸在初始位（自检）, #3腔体平移气缸在氦检位（自检）, #3腔体抽真空阀状态（自检）, #3腔体破真空阀状态（自检）, #3腔体抽气阀打开允许（自检）, #3腔体自检停止(SW), #3腔体自检启动(SW), #3腔体机构复位（M）, #3氦检机构初始位, #3-1腔体单腔自检(SW), #3-2腔体单腔自检(SW), #3腔体自检运行中, #3-1腔体自检保压前真空（Pa_Float）, #3-1腔体自检保压后真空（Pa_Float）, #3-1腔体自检泄漏量（Pa_Float）, #3-1腔体自检结果（1-OK，2-NG）, #3腔体真空泵开（自检）, #3腔体平移气缸到初始位（自检）, #3腔体平移气缸到氦检位（自检）, #3腔体顶升气缸下降（自检）, #3腔体顶升气缸上升（自检）, #3腔体开抽真空阀（自检）, #3腔体关抽真空阀（自检）, #3腔体开破真空阀（自检）, #3腔体关破真空阀（自检）, #3-1腔体自检前保压时间（S_UInt）, #3-1腔体自检保压时间（S_UInt）, #3-1腔体自检抽气时间（S_UInt）, #3腔体抽气阀打开需求（自检）, #3-2腔体自检保压前真空（Pa_Float）, #3-2腔体自检保压后真空（Pa_Float）, #3-2腔体自检泄漏量（Pa_Float）, #3-2腔体自检结果（1-OK，2-NG,3-抽真空NG）, #3-2腔体自检前保压时间（S_UInt）, #3-2腔体自检保压时间（S_UInt）, #3-2腔体自检抽气时间（S_UInt）

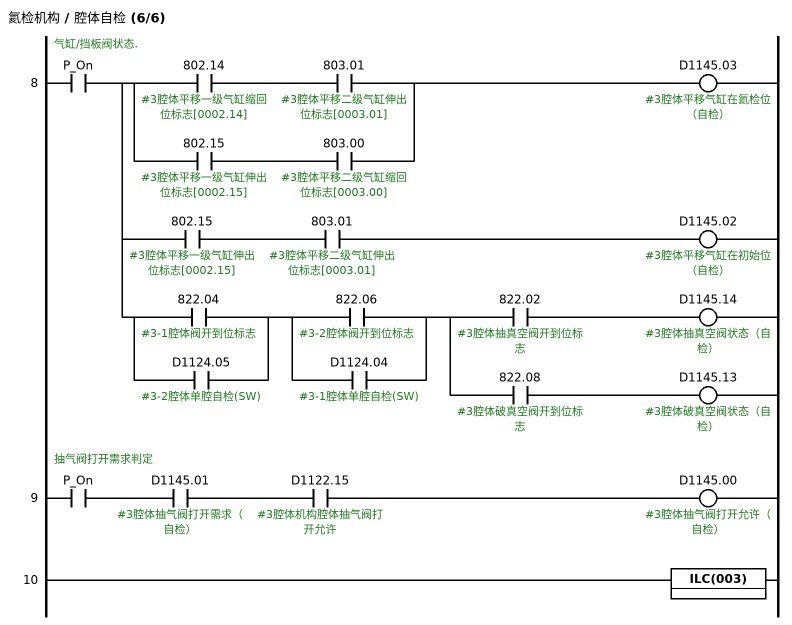
; rung 8: 气缸/挡板阀状态.
LD P_On
OUT TR0
LD 802.14  ; #3腔体平移一级气缸缩回位标志[0002.14]
AND 803.01  ; #3腔体平移二级气缸伸出位标志[0003.01]
LD 802.15  ; #3腔体平移一级气缸伸出位标志[0002.15]
AND 803.00  ; #3腔体平移二级气缸缩回位标志[0003.00]
ORLD
ANDLD
OUT D1145.03  ; #3腔体平移气缸在氦检位（自检）
LD TR0
AND 802.15  ; #3腔体平移一级气缸伸出位标志[0002.15]
AND 803.01  ; #3腔体平移二级气缸伸出位标志[0003.01]
OUT D1145.02  ; #3腔体平移气缸在初始位（自检）
LD TR0
LD 822.04  ; #3-1腔体阀开到位标志
OR D1124.05  ; #3-2腔体单腔自检(SW)
ANDLD
LD 822.06  ; #3-2腔体阀开到位标志
OR D1124.04  ; #3-1腔体单腔自检(SW)
ANDLD
OUT TR0
AND 822.02  ; #3腔体抽真空阀开到位标志
OUT D1145.14  ; #3腔体抽真空阀状态（自检）
LD TR0
AND 822.08  ; #3腔体破真空阀开到位标志
OUT D1145.13  ; #3腔体破真空阀状态（自检）
; rung 9: 抽气阀打开需求判定
LD P_On
AND D1145.01  ; #3腔体抽气阀打开需求（自检）
AND D1122.15  ; #3腔体机构腔体抽气阀打开允许
OUT D1145.00  ; #3腔体抽气阀打开允许（自检）
; rung 10
ILC(003)

### Section 指示灯

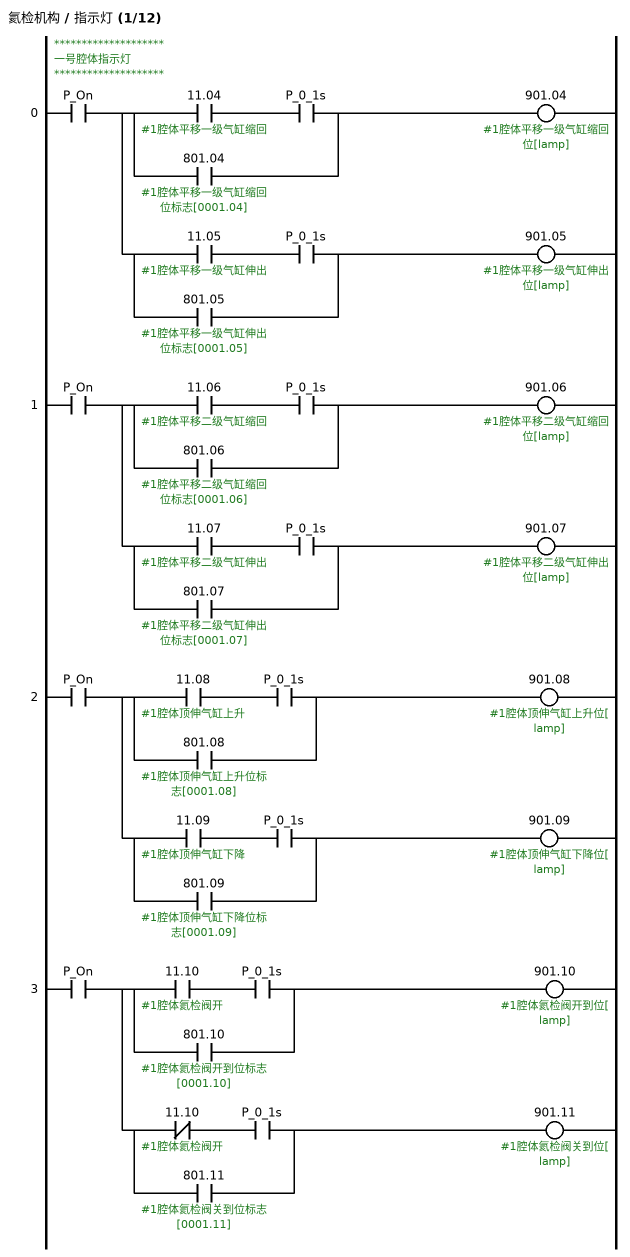
; rung 0: ******************** / 一号腔体指示灯 / ********************
LD P_On
OUT TR0
LD 11.04  ; #1腔体平移一级气缸缩回
AND P_0_1s
OR 801.04  ; #1腔体平移一级气缸缩回位标志[0001.04]
ANDLD
OUT 901.04  ; #1腔体平移一级气缸缩回位[lamp]
LD TR0
LD 11.05  ; #1腔体平移一级气缸伸出
AND P_0_1s
OR 801.05  ; #1腔体平移一级气缸伸出位标志[0001.05]
ANDLD
OUT 901.05  ; #1腔体平移一级气缸伸出位[lamp]
; rung 1
LD P_On
OUT TR0
LD 11.06  ; #1腔体平移二级气缸缩回
AND P_0_1s
OR 801.06  ; #1腔体平移二级气缸缩回位标志[0001.06]
ANDLD
OUT 901.06  ; #1腔体平移二级气缸缩回位[lamp]
LD TR0
LD 11.07  ; #1腔体平移二级气缸伸出
AND P_0_1s
OR 801.07  ; #1腔体平移二级气缸伸出位标志[0001.07]
ANDLD
OUT 901.07  ; #1腔体平移二级气缸伸出位[lamp]
; rung 2
LD P_On
OUT TR0
LD 11.08  ; #1腔体顶伸气缸上升
AND P_0_1s
OR 801.08  ; #1腔体顶伸气缸上升位标志[0001.08]
ANDLD
OUT 901.08  ; #1腔体顶伸气缸上升位[lamp]
LD TR0
LD 11.09  ; #1腔体顶伸气缸下降
AND P_0_1s
OR 801.09  ; #1腔体顶伸气缸下降位标志[0001.09]
ANDLD
OUT 901.09  ; #1腔体顶伸气缸下降位[lamp]
; rung 3
LD P_On
OUT TR0
LD 11.10  ; #1腔体氦检阀开
AND P_0_1s
OR 801.10  ; #1腔体氦检阀开到位标志[0001.10]
ANDLD
OUT 901.10  ; #1腔体氦检阀开到位[lamp]
LD TR0
LDNOT 11.10  ; #1腔体氦检阀开
AND P_0_1s
OR 801.11  ; #1腔体氦检阀关到位标志[0001.11]
ANDLD
OUT 901.11  ; #1腔体氦检阀关到位[lamp]

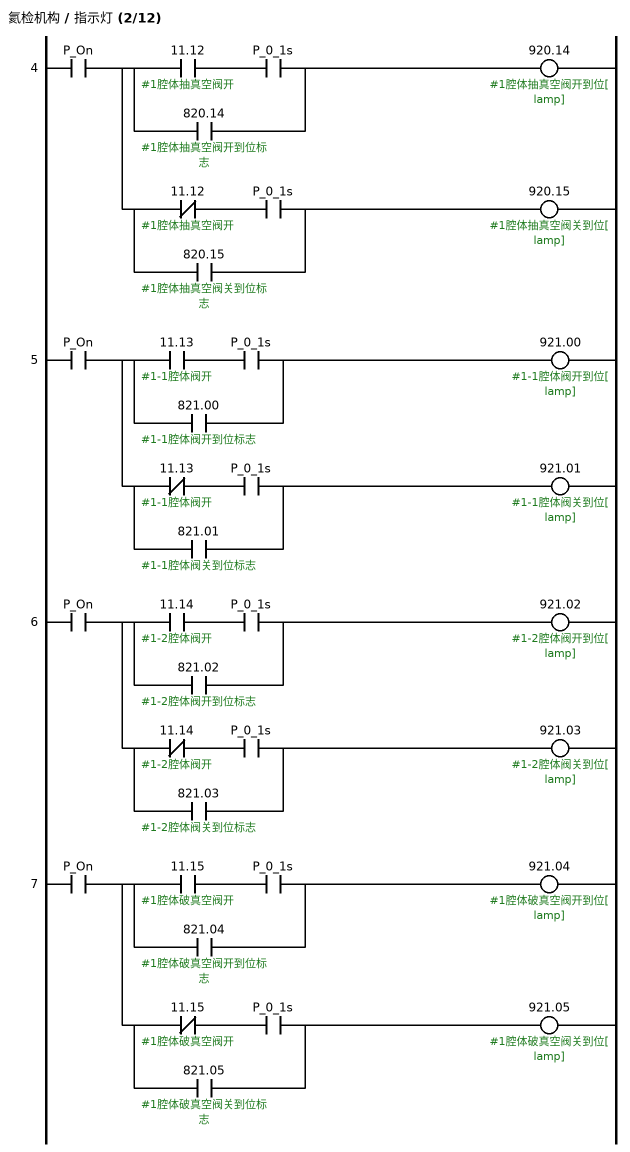
; rung 4
LD P_On
OUT TR0
LD 11.12  ; #1腔体抽真空阀开
AND P_0_1s
OR 820.14  ; #1腔体抽真空阀开到位标志
ANDLD
OUT 920.14  ; #1腔体抽真空阀开到位[lamp]
LD TR0
LDNOT 11.12  ; #1腔体抽真空阀开
AND P_0_1s
OR 820.15  ; #1腔体抽真空阀关到位标志
ANDLD
OUT 920.15  ; #1腔体抽真空阀关到位[lamp]
; rung 5
LD P_On
OUT TR0
LD 11.13  ; #1-1腔体阀开
AND P_0_1s
OR 821.00  ; #1-1腔体阀开到位标志
ANDLD
OUT 921.00  ; #1-1腔体阀开到位[lamp]
LD TR0
LDNOT 11.13  ; #1-1腔体阀开
AND P_0_1s
OR 821.01  ; #1-1腔体阀关到位标志
ANDLD
OUT 921.01  ; #1-1腔体阀关到位[lamp]
; rung 6
LD P_On
OUT TR0
LD 11.14  ; #1-2腔体阀开
AND P_0_1s
OR 821.02  ; #1-2腔体阀开到位标志
ANDLD
OUT 921.02  ; #1-2腔体阀开到位[lamp]
LD TR0
LDNOT 11.14  ; #1-2腔体阀开
AND P_0_1s
OR 821.03  ; #1-2腔体阀关到位标志
ANDLD
OUT 921.03  ; #1-2腔体阀关到位[lamp]
; rung 7
LD P_On
OUT TR0
LD 11.15  ; #1腔体破真空阀开
AND P_0_1s
OR 821.04  ; #1腔体破真空阀开到位标志
ANDLD
OUT 921.04  ; #1腔体破真空阀开到位[lamp]
LD TR0
LDNOT 11.15  ; #1腔体破真空阀开
AND P_0_1s
OR 821.05  ; #1腔体破真空阀关到位标志
ANDLD
OUT 921.05  ; #1腔体破真空阀关到位[lamp]

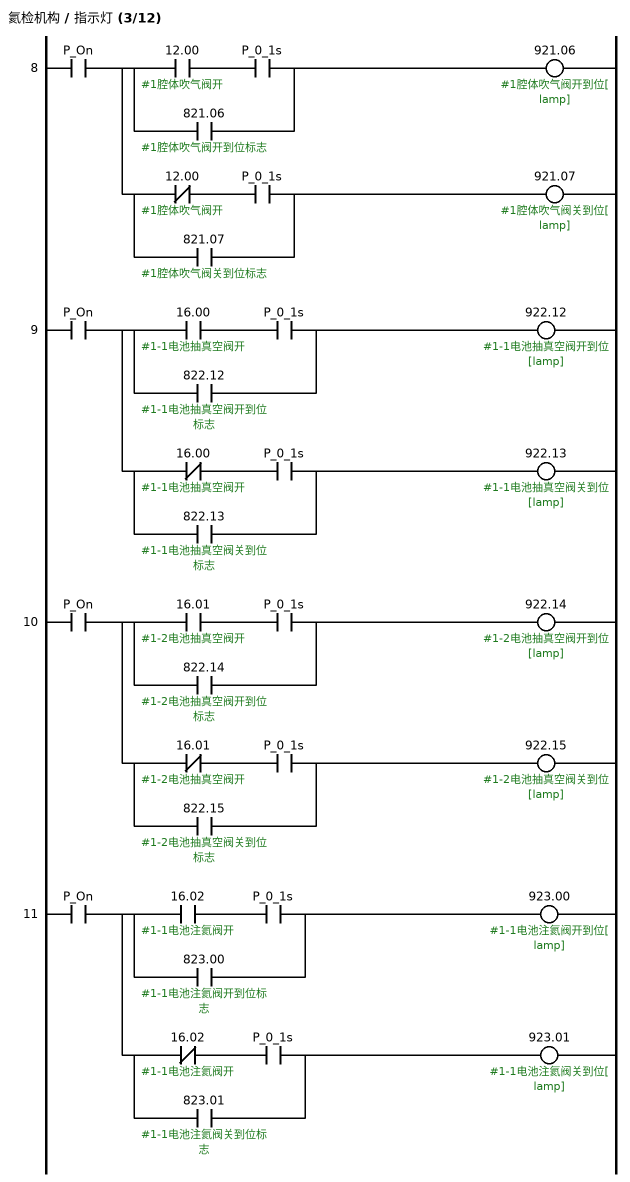
; rung 8
LD P_On
OUT TR0
LD 12.00  ; #1腔体吹气阀开
AND P_0_1s
OR 821.06  ; #1腔体吹气阀开到位标志
ANDLD
OUT 921.06  ; #1腔体吹气阀开到位[lamp]
LD TR0
LDNOT 12.00  ; #1腔体吹气阀开
AND P_0_1s
OR 821.07  ; #1腔体吹气阀关到位标志
ANDLD
OUT 921.07  ; #1腔体吹气阀关到位[lamp]
; rung 9
LD P_On
OUT TR0
LD 16.00  ; #1-1电池抽真空阀开
AND P_0_1s
OR 822.12  ; #1-1电池抽真空阀开到位标志
ANDLD
OUT 922.12  ; #1-1电池抽真空阀开到位[lamp]
LD TR0
LDNOT 16.00  ; #1-1电池抽真空阀开
AND P_0_1s
OR 822.13  ; #1-1电池抽真空阀关到位标志
ANDLD
OUT 922.13  ; #1-1电池抽真空阀关到位[lamp]
; rung 10
LD P_On
OUT TR0
LD 16.01  ; #1-2电池抽真空阀开
AND P_0_1s
OR 822.14  ; #1-2电池抽真空阀开到位标志
ANDLD
OUT 922.14  ; #1-2电池抽真空阀开到位[lamp]
LD TR0
LDNOT 16.01  ; #1-2电池抽真空阀开
AND P_0_1s
OR 822.15  ; #1-2电池抽真空阀关到位标志
ANDLD
OUT 922.15  ; #1-2电池抽真空阀关到位[lamp]
; rung 11
LD P_On
OUT TR0
LD 16.02  ; #1-1电池注氦阀开
AND P_0_1s
OR 823.00  ; #1-1电池注氦阀开到位标志
ANDLD
OUT 923.00  ; #1-1电池注氦阀开到位[lamp]
LD TR0
LDNOT 16.02  ; #1-1电池注氦阀开
AND P_0_1s
OR 823.01  ; #1-1电池注氦阀关到位标志
ANDLD
OUT 923.01  ; #1-1电池注氦阀关到位[lamp]

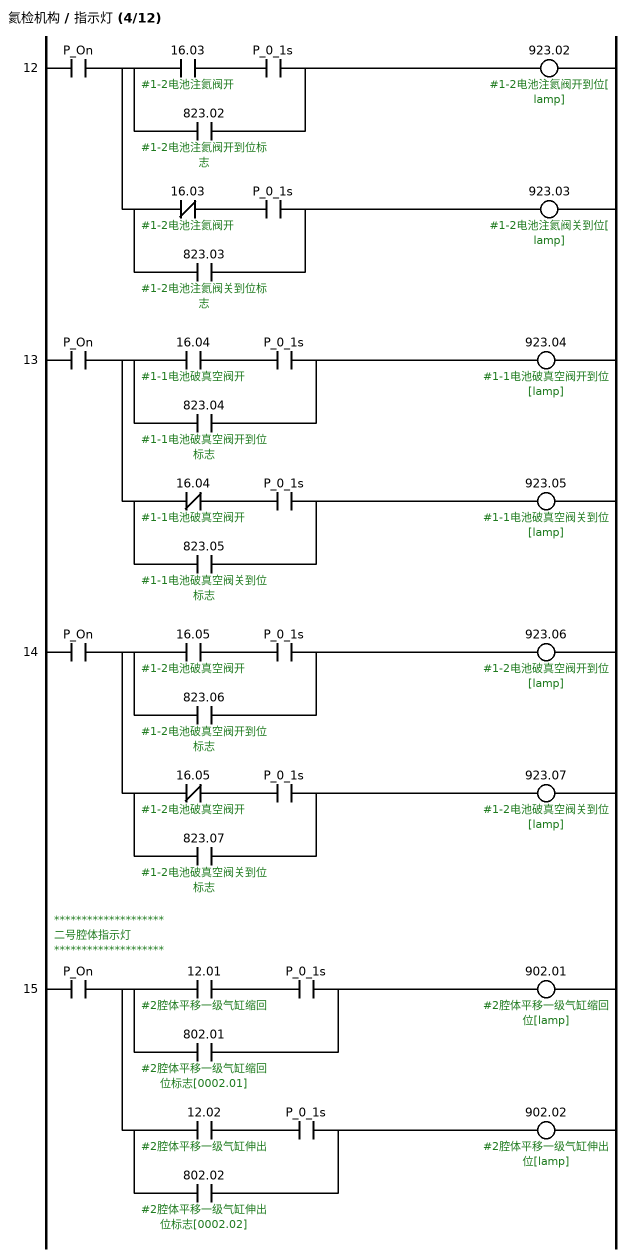
; rung 12
LD P_On
OUT TR0
LD 16.03  ; #1-2电池注氦阀开
AND P_0_1s
OR 823.02  ; #1-2电池注氦阀开到位标志
ANDLD
OUT 923.02  ; #1-2电池注氦阀开到位[lamp]
LD TR0
LDNOT 16.03  ; #1-2电池注氦阀开
AND P_0_1s
OR 823.03  ; #1-2电池注氦阀关到位标志
ANDLD
OUT 923.03  ; #1-2电池注氦阀关到位[lamp]
; rung 13
LD P_On
OUT TR0
LD 16.04  ; #1-1电池破真空阀开
AND P_0_1s
OR 823.04  ; #1-1电池破真空阀开到位标志
ANDLD
OUT 923.04  ; #1-1电池破真空阀开到位[lamp]
LD TR0
LDNOT 16.04  ; #1-1电池破真空阀开
AND P_0_1s
OR 823.05  ; #1-1电池破真空阀关到位标志
ANDLD
OUT 923.05  ; #1-1电池破真空阀关到位[lamp]
; rung 14
LD P_On
OUT TR0
LD 16.05  ; #1-2电池破真空阀开
AND P_0_1s
OR 823.06  ; #1-2电池破真空阀开到位标志
ANDLD
OUT 923.06  ; #1-2电池破真空阀开到位[lamp]
LD TR0
LDNOT 16.05  ; #1-2电池破真空阀开
AND P_0_1s
OR 823.07  ; #1-2电池破真空阀关到位标志
ANDLD
OUT 923.07  ; #1-2电池破真空阀关到位[lamp]
; rung 15: ******************** / 二号腔体指示灯 / ********************
LD P_On
OUT TR0
LD 12.01  ; #2腔体平移一级气缸缩回
AND P_0_1s
OR 802.01  ; #2腔体平移一级气缸缩回位标志[0002.01]
ANDLD
OUT 902.01  ; #2腔体平移一级气缸缩回位[lamp]
LD TR0
LD 12.02  ; #2腔体平移一级气缸伸出
AND P_0_1s
OR 802.02  ; #2腔体平移一级气缸伸出位标志[0002.02]
ANDLD
OUT 902.02  ; #2腔体平移一级气缸伸出位[lamp]

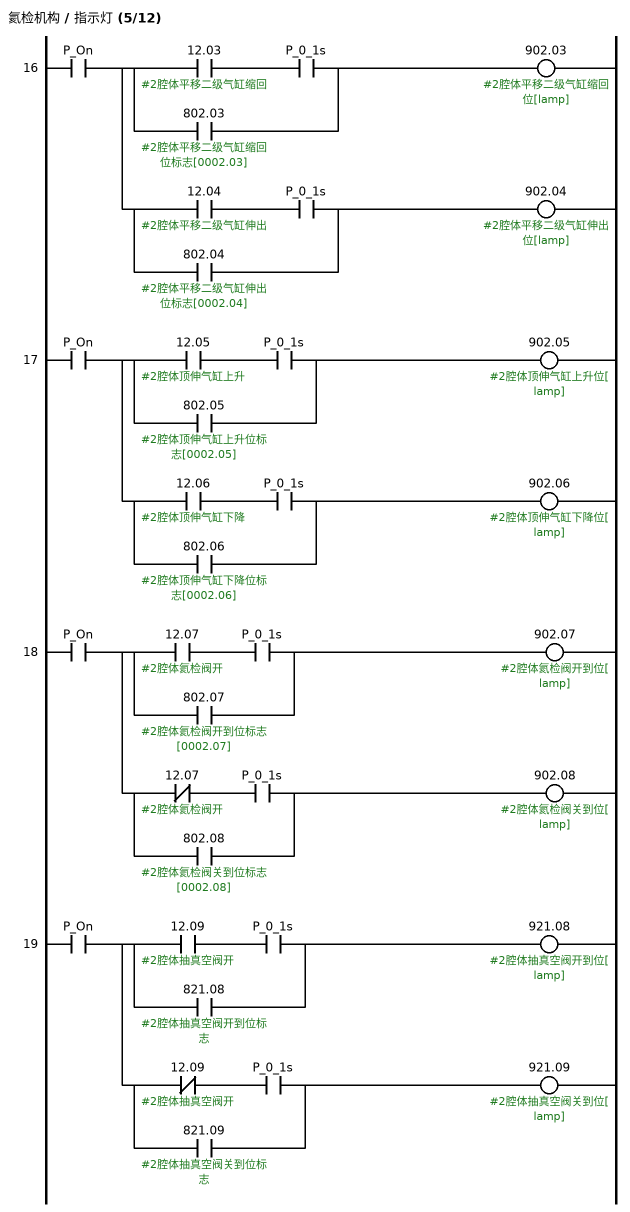
; rung 16
LD P_On
OUT TR0
LD 12.03  ; #2腔体平移二级气缸缩回
AND P_0_1s
OR 802.03  ; #2腔体平移二级气缸缩回位标志[0002.03]
ANDLD
OUT 902.03  ; #2腔体平移二级气缸缩回位[lamp]
LD TR0
LD 12.04  ; #2腔体平移二级气缸伸出
AND P_0_1s
OR 802.04  ; #2腔体平移二级气缸伸出位标志[0002.04]
ANDLD
OUT 902.04  ; #2腔体平移二级气缸伸出位[lamp]
; rung 17
LD P_On
OUT TR0
LD 12.05  ; #2腔体顶伸气缸上升
AND P_0_1s
OR 802.05  ; #2腔体顶伸气缸上升位标志[0002.05]
ANDLD
OUT 902.05  ; #2腔体顶伸气缸上升位[lamp]
LD TR0
LD 12.06  ; #2腔体顶伸气缸下降
AND P_0_1s
OR 802.06  ; #2腔体顶伸气缸下降位标志[0002.06]
ANDLD
OUT 902.06  ; #2腔体顶伸气缸下降位[lamp]
; rung 18
LD P_On
OUT TR0
LD 12.07  ; #2腔体氦检阀开
AND P_0_1s
OR 802.07  ; #2腔体氦检阀开到位标志[0002.07]
ANDLD
OUT 902.07  ; #2腔体氦检阀开到位[lamp]
LD TR0
LDNOT 12.07  ; #2腔体氦检阀开
AND P_0_1s
OR 802.08  ; #2腔体氦检阀关到位标志[0002.08]
ANDLD
OUT 902.08  ; #2腔体氦检阀关到位[lamp]
; rung 19
LD P_On
OUT TR0
LD 12.09  ; #2腔体抽真空阀开
AND P_0_1s
OR 821.08  ; #2腔体抽真空阀开到位标志
ANDLD
OUT 921.08  ; #2腔体抽真空阀开到位[lamp]
LD TR0
LDNOT 12.09  ; #2腔体抽真空阀开
AND P_0_1s
OR 821.09  ; #2腔体抽真空阀关到位标志
ANDLD
OUT 921.09  ; #2腔体抽真空阀关到位[lamp]

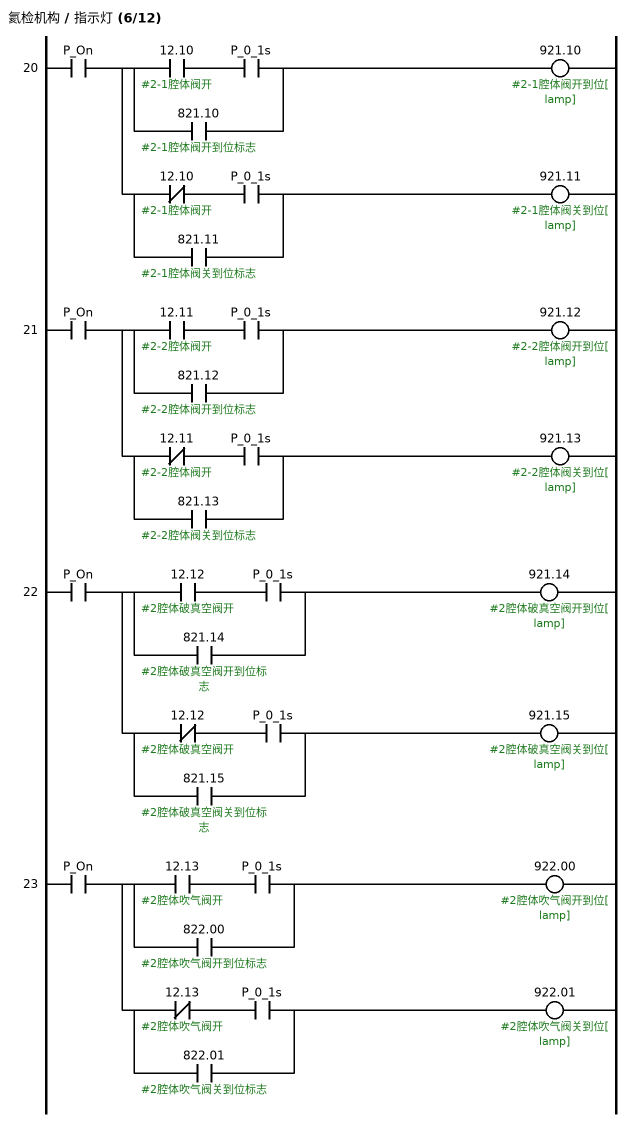
; rung 20
LD P_On
OUT TR0
LD 12.10  ; #2-1腔体阀开
AND P_0_1s
OR 821.10  ; #2-1腔体阀开到位标志
ANDLD
OUT 921.10  ; #2-1腔体阀开到位[lamp]
LD TR0
LDNOT 12.10  ; #2-1腔体阀开
AND P_0_1s
OR 821.11  ; #2-1腔体阀关到位标志
ANDLD
OUT 921.11  ; #2-1腔体阀关到位[lamp]
; rung 21
LD P_On
OUT TR0
LD 12.11  ; #2-2腔体阀开
AND P_0_1s
OR 821.12  ; #2-2腔体阀开到位标志
ANDLD
OUT 921.12  ; #2-2腔体阀开到位[lamp]
LD TR0
LDNOT 12.11  ; #2-2腔体阀开
AND P_0_1s
OR 821.13  ; #2-2腔体阀关到位标志
ANDLD
OUT 921.13  ; #2-2腔体阀关到位[lamp]
; rung 22
LD P_On
OUT TR0
LD 12.12  ; #2腔体破真空阀开
AND P_0_1s
OR 821.14  ; #2腔体破真空阀开到位标志
ANDLD
OUT 921.14  ; #2腔体破真空阀开到位[lamp]
LD TR0
LDNOT 12.12  ; #2腔体破真空阀开
AND P_0_1s
OR 821.15  ; #2腔体破真空阀关到位标志
ANDLD
OUT 921.15  ; #2腔体破真空阀关到位[lamp]
; rung 23
LD P_On
OUT TR0
LD 12.13  ; #2腔体吹气阀开
AND P_0_1s
OR 822.00  ; #2腔体吹气阀开到位标志
ANDLD
OUT 922.00  ; #2腔体吹气阀开到位[lamp]
LD TR0
LDNOT 12.13  ; #2腔体吹气阀开
AND P_0_1s
OR 822.01  ; #2腔体吹气阀关到位标志
ANDLD
OUT 922.01  ; #2腔体吹气阀关到位[lamp]

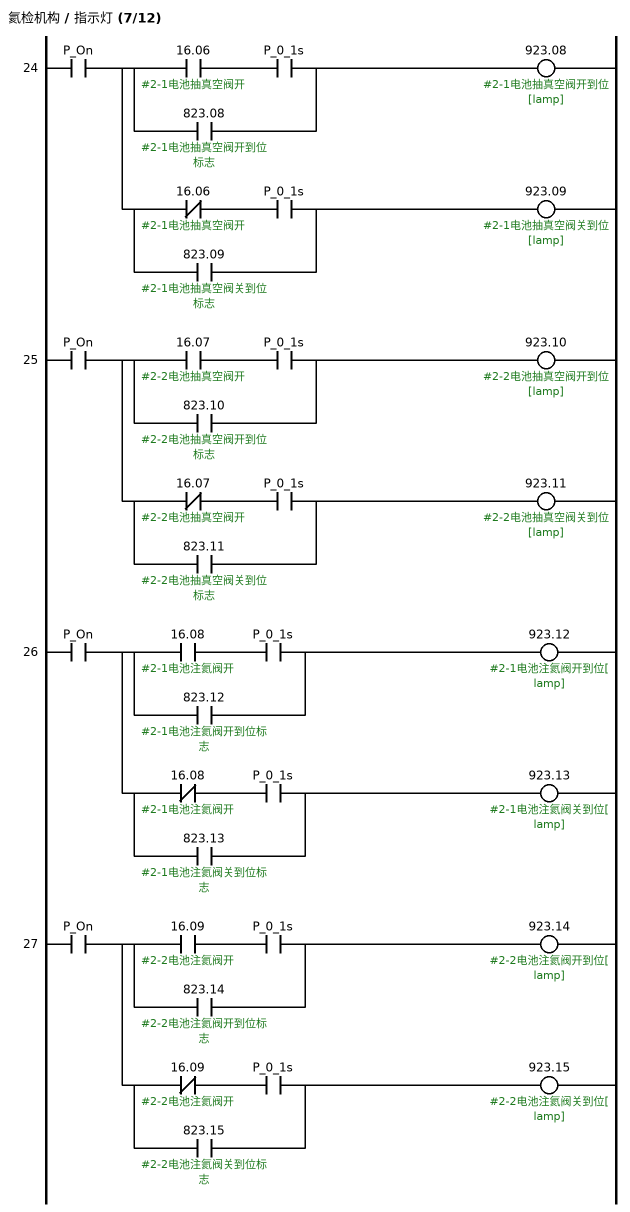
; rung 24
LD P_On
OUT TR0
LD 16.06  ; #2-1电池抽真空阀开
AND P_0_1s
OR 823.08  ; #2-1电池抽真空阀开到位标志
ANDLD
OUT 923.08  ; #2-1电池抽真空阀开到位[lamp]
LD TR0
LDNOT 16.06  ; #2-1电池抽真空阀开
AND P_0_1s
OR 823.09  ; #2-1电池抽真空阀关到位标志
ANDLD
OUT 923.09  ; #2-1电池抽真空阀关到位[lamp]
; rung 25
LD P_On
OUT TR0
LD 16.07  ; #2-2电池抽真空阀开
AND P_0_1s
OR 823.10  ; #2-2电池抽真空阀开到位标志
ANDLD
OUT 923.10  ; #2-2电池抽真空阀开到位[lamp]
LD TR0
LDNOT 16.07  ; #2-2电池抽真空阀开
AND P_0_1s
OR 823.11  ; #2-2电池抽真空阀关到位标志
ANDLD
OUT 923.11  ; #2-2电池抽真空阀关到位[lamp]
; rung 26
LD P_On
OUT TR0
LD 16.08  ; #2-1电池注氦阀开
AND P_0_1s
OR 823.12  ; #2-1电池注氦阀开到位标志
ANDLD
OUT 923.12  ; #2-1电池注氦阀开到位[lamp]
LD TR0
LDNOT 16.08  ; #2-1电池注氦阀开
AND P_0_1s
OR 823.13  ; #2-1电池注氦阀关到位标志
ANDLD
OUT 923.13  ; #2-1电池注氦阀关到位[lamp]
; rung 27
LD P_On
OUT TR0
LD 16.09  ; #2-2电池注氦阀开
AND P_0_1s
OR 823.14  ; #2-2电池注氦阀开到位标志
ANDLD
OUT 923.14  ; #2-2电池注氦阀开到位[lamp]
LD TR0
LDNOT 16.09  ; #2-2电池注氦阀开
AND P_0_1s
OR 823.15  ; #2-2电池注氦阀关到位标志
ANDLD
OUT 923.15  ; #2-2电池注氦阀关到位[lamp]

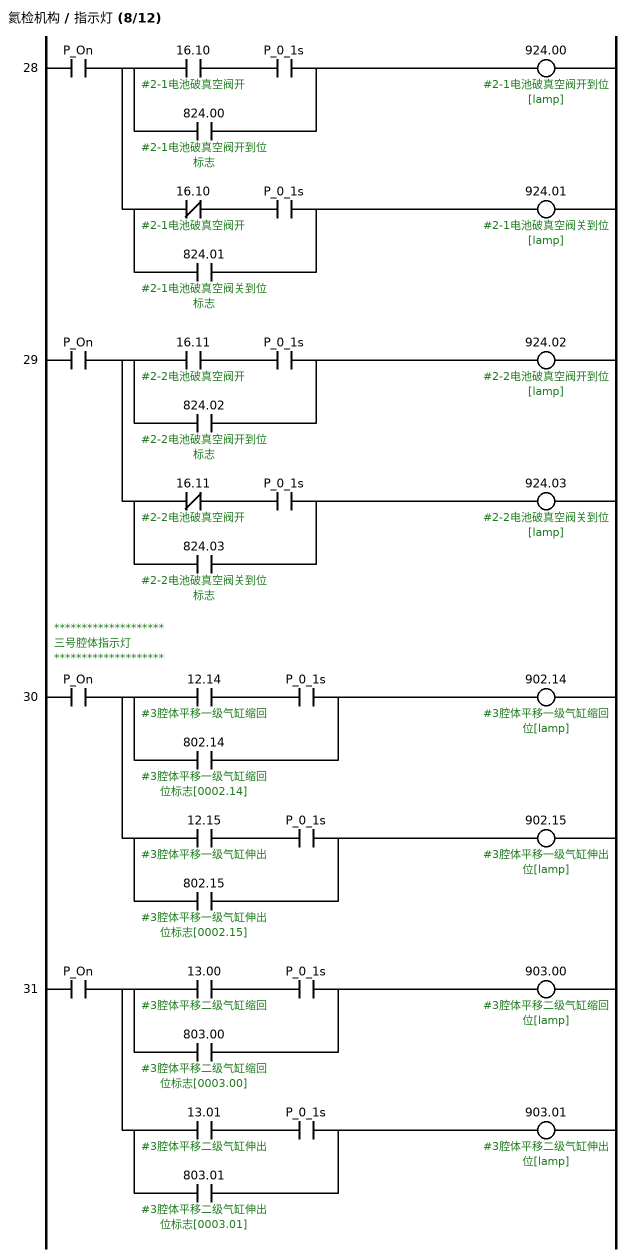
; rung 28
LD P_On
OUT TR0
LD 16.10  ; #2-1电池破真空阀开
AND P_0_1s
OR 824.00  ; #2-1电池破真空阀开到位标志
ANDLD
OUT 924.00  ; #2-1电池破真空阀开到位[lamp]
LD TR0
LDNOT 16.10  ; #2-1电池破真空阀开
AND P_0_1s
OR 824.01  ; #2-1电池破真空阀关到位标志
ANDLD
OUT 924.01  ; #2-1电池破真空阀关到位[lamp]
; rung 29
LD P_On
OUT TR0
LD 16.11  ; #2-2电池破真空阀开
AND P_0_1s
OR 824.02  ; #2-2电池破真空阀开到位标志
ANDLD
OUT 924.02  ; #2-2电池破真空阀开到位[lamp]
LD TR0
LDNOT 16.11  ; #2-2电池破真空阀开
AND P_0_1s
OR 824.03  ; #2-2电池破真空阀关到位标志
ANDLD
OUT 924.03  ; #2-2电池破真空阀关到位[lamp]
; rung 30: ******************** / 三号腔体指示灯 / ********************
LD P_On
OUT TR0
LD 12.14  ; #3腔体平移一级气缸缩回
AND P_0_1s
OR 802.14  ; #3腔体平移一级气缸缩回位标志[0002.14]
ANDLD
OUT 902.14  ; #3腔体平移一级气缸缩回位[lamp]
LD TR0
LD 12.15  ; #3腔体平移一级气缸伸出
AND P_0_1s
OR 802.15  ; #3腔体平移一级气缸伸出位标志[0002.15]
ANDLD
OUT 902.15  ; #3腔体平移一级气缸伸出位[lamp]
; rung 31
LD P_On
OUT TR0
LD 13.00  ; #3腔体平移二级气缸缩回
AND P_0_1s
OR 803.00  ; #3腔体平移二级气缸缩回位标志[0003.00]
ANDLD
OUT 903.00  ; #3腔体平移二级气缸缩回位[lamp]
LD TR0
LD 13.01  ; #3腔体平移二级气缸伸出
AND P_0_1s
OR 803.01  ; #3腔体平移二级气缸伸出位标志[0003.01]
ANDLD
OUT 903.01  ; #3腔体平移二级气缸伸出位[lamp]

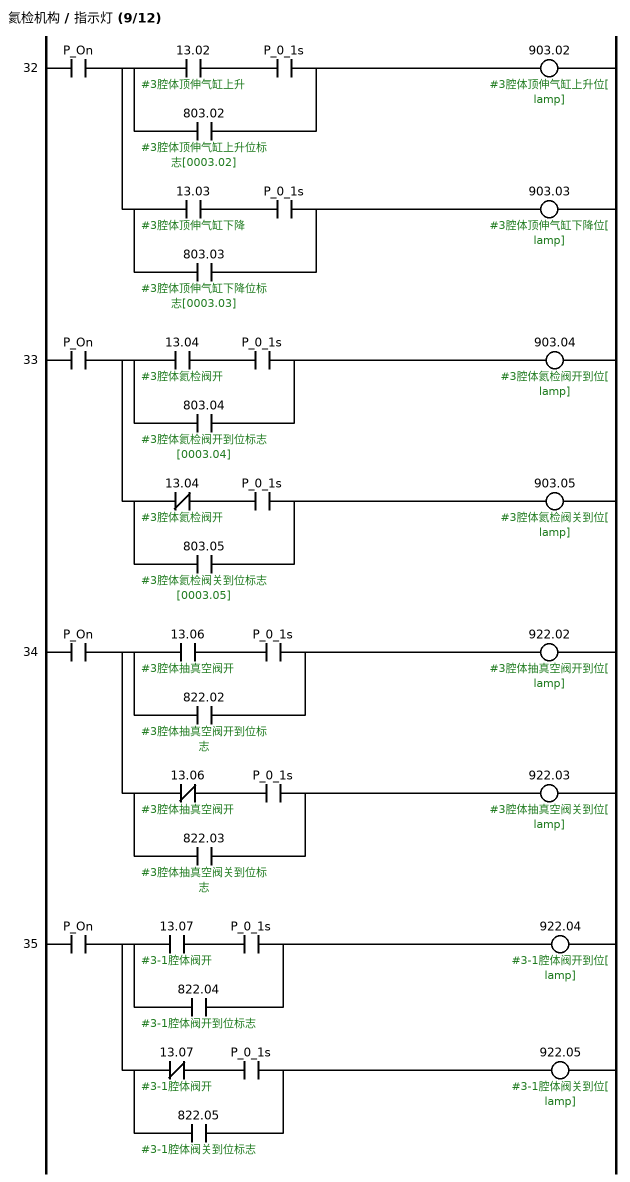
; rung 32
LD P_On
OUT TR0
LD 13.02  ; #3腔体顶伸气缸上升
AND P_0_1s
OR 803.02  ; #3腔体顶伸气缸上升位标志[0003.02]
ANDLD
OUT 903.02  ; #3腔体顶伸气缸上升位[lamp]
LD TR0
LD 13.03  ; #3腔体顶伸气缸下降
AND P_0_1s
OR 803.03  ; #3腔体顶伸气缸下降位标志[0003.03]
ANDLD
OUT 903.03  ; #3腔体顶伸气缸下降位[lamp]
; rung 33
LD P_On
OUT TR0
LD 13.04  ; #3腔体氦检阀开
AND P_0_1s
OR 803.04  ; #3腔体氦检阀开到位标志[0003.04]
ANDLD
OUT 903.04  ; #3腔体氦检阀开到位[lamp]
LD TR0
LDNOT 13.04  ; #3腔体氦检阀开
AND P_0_1s
OR 803.05  ; #3腔体氦检阀关到位标志[0003.05]
ANDLD
OUT 903.05  ; #3腔体氦检阀关到位[lamp]
; rung 34
LD P_On
OUT TR0
LD 13.06  ; #3腔体抽真空阀开
AND P_0_1s
OR 822.02  ; #3腔体抽真空阀开到位标志
ANDLD
OUT 922.02  ; #3腔体抽真空阀开到位[lamp]
LD TR0
LDNOT 13.06  ; #3腔体抽真空阀开
AND P_0_1s
OR 822.03  ; #3腔体抽真空阀关到位标志
ANDLD
OUT 922.03  ; #3腔体抽真空阀关到位[lamp]
; rung 35
LD P_On
OUT TR0
LD 13.07  ; #3-1腔体阀开
AND P_0_1s
OR 822.04  ; #3-1腔体阀开到位标志
ANDLD
OUT 922.04  ; #3-1腔体阀开到位[lamp]
LD TR0
LDNOT 13.07  ; #3-1腔体阀开
AND P_0_1s
OR 822.05  ; #3-1腔体阀关到位标志
ANDLD
OUT 922.05  ; #3-1腔体阀关到位[lamp]

